CASE _Scenario OF
	QUEUE_CLEANUP_TEST_SCENARIO.REPEATED_EXECUTE_FAILURE:
		_Child.CleanupFailures := 2;
		_ExpectedExecuteFailures := 3;

	QUEUE_CLEANUP_TEST_SCENARIO.CANCEL_REQUEST_FAILURE:
		_Child.CancelFailures := 2;
		_ExpectedCancelFailures := 2;

	QUEUE_CLEANUP_TEST_SCENARIO.MESSAGE_FORMATTING_FAILURE:
		_ExpectedFailureMessage := "Task 'queue' processing failed";
END_CASE

_Resource.SetChild(child := _Child);
_Resource.SetThrowOnStartRelease(throwOnStartRelease := _InjectReleaseFailure);
_Queue.SetResourceManager(resourceManager := _Resource);
_Queue.StopWhenNoPendingTasks := TRUE;
_Queue.Enqueue(task := _Child);
_Queue.Enqueue(task := _Waiting);
Assert.ThatBool(actual := _Queue.Start(), message := "Prepared queue must accept Start").IsTrue();
END_METHOD

(*!
<summary>Advances one queue call and observes the selected failure or reuse case.</summary>
<description>
An escaping exception uses the framework's ExecuteTest diagnostic and proceeds to AfterTest.
</description>
*)
METHOD PROTECTED ExecuteTest : TOF_Testing.TEST_CYCLE_RESULT
ExecuteTest := TOF_Testing.TEST_CYCLE_RESULT.DONE;

IF CycleCount - _RunStartCycle > _MaxRunCycles THEN
	RecordFailure(message := "Queue cleanup or reuse exceeded its cycle budget");
	RETURN;
END_IF

_Queue.Execute();

CASE _Phase OF
	QUEUE_CLEANUP_TEST_PHASE.REUSE_RUN:
		IF _Queue.State.Stopped THEN
			checkSuccessfulReuse();
		ELSE
			ExecuteTest := TOF_Testing.TEST_CYCLE_RESULT.BUSY;
		END_IF

	QUEUE_CLEANUP_TEST_PHASE.OBSERVE_FAILED_RELEASE:
		Assert.ThatBool(
			actual := _Queue.State.Stopped AND_THEN _Queue.FinalStopReason.Failure,
			message := "Failed release must leave the queue stopped"
		).IsTrue();
		Assert.ThatUInt(
			actual := _Resource.ReleaseCalls,
			message := "A stopped queue must not retry a failed release"
		).ToBe(expected := 1);
		Assert.ThatBool(
			actual := _Resource.ResourceAcquired,
			message := "The failed release must leave the synthetic resource held"
		).IsTrue();

	QUEUE_CLEANUP_TEST_PHASE.FAILURE_RUN:
		IF NOT _Queue.State.Stopped THEN
			IF _Child.ExecuteFailuresRaised > 0 THEN
				observePendingFailure();
			END_IF

			ExecuteTest := TOF_Testing.TEST_CYCLE_RESULT.BUSY;
			RETURN;
		END_IF

		checkFailedRun();

		IF Outcome = TOF_Testing.TEST_OUTCOME.FAILED THEN
			RETURN;
		END_IF

		IF _Scenario = QUEUE_CLEANUP_TEST_SCENARIO.DELAYED_CLEANUP_AND_REUSE THEN
			IF startReuse() THEN
				_Phase := QUEUE_CLEANUP_TEST_PHASE.REUSE_RUN;
				_RunStartCycle := CycleCount;
				ExecuteTest := TOF_Testing.TEST_CYCLE_RESULT.BUSY;
			END_IF
		ELSIF _InjectReleaseFailure THEN
			_Phase := QUEUE_CLEANUP_TEST_PHASE.OBSERVE_FAILED_RELEASE;
			ExecuteTest := TOF_Testing.TEST_CYCLE_RESULT.BUSY;
		END_IF
END_CASE
END_METHOD

(*!
<summary>Checks ownership while the failed current child is still running.</summary>
<description>
On the initial failure call, confirms cleanup was deferred and optionally requests owner cancellation.
For held cleanup, counts subsequent queue calls before allowing the child to finish.
</description>
*)
METHOD PRIVATE observePendingFailure
IF NOT _Child.State.Running THEN
	RETURN;
END_IF

Assert.ThatBool(
	actual := _Queue.State.Running AND_THEN _Queue.RunningSubstate.Stopping,
	message := "The queue must wait in STOPPING for the child"
).IsTrue();
Assert.ThatBool(
	actual := _Resource.ResourceAcquired,
	message := "The queue must retain its resource during child cleanup"
).IsTrue();
Assert.ThatUInt(
	actual := _Resource.ReleaseCalls,
	message := "Release must wait for child cleanup"
).ToBe(expected := 0);
Assert.ThatBool(
	actual := _Waiting.State.Ready,
	message := "Waiting child must remain READY during cleanup"
).IsTrue();

IF NOT _FirstFailureObserved THEN
	_FirstFailureObserved := TRUE;
	Assert.ThatBool(
		actual := _Queue.OriginalStopReason.Failure,
		message := "The initial Execute exception must set the original result to FAILURE"
	).IsTrue();
	Assert.ThatUInt(
		actual := _Child.CompletedCleanupSteps,
		message := "The call that failed must not advance child cleanup"
	).ToBe(expected := 0);

	IF _RequestExternalCancel THEN
		Assert.ThatWideString(
			actual := _Queue.OriginalStopReason.Message,
			message := "Observe the first child failure before owner cancellation"
		).ToBe(expected := _ExpectedFailureMessage);
		Assert.ThatBool(
			actual := _Queue.Cancel(),
			message := "Owner Cancel must be accepted while failure cleanup is pending"
		).IsTrue();
		Assert.ThatBool(
			actual := _Queue.OriginalStopReason.ExternalCancel,
			message := "Accepted Cancel must replace the original failure reason"
		).IsTrue();
	END_IF

	RETURN;
END_IF

IF _Child.HoldCleanup THEN
	_HeldCycles := _HeldCycles + 1;
	Assert.ThatUInt(
		actual := _Child.CompletedCleanupSteps,
		message := "Held cleanup must not advance"
	).ToBe(expected := 0);

	IF _HeldCycles = _HeldObservationCycles THEN
		_Child.HoldCleanup := FALSE;
	END_IF
END_IF
END_METHOD

(*!
<summary>Checks the stopped queue, fault counts, entry ownership and release ordering.</summary>
*)
METHOD PRIVATE checkFailedRun
Assert.ThatBool(
	actual := _FirstFailureObserved,
	message := "Observe the initial failure while the child is RUNNING"
).IsTrue();
Assert.ThatBool(
	actual := _Child.State.Stopped,
	message := "Parent must not stop ahead of the failed child"
).IsTrue();
Assert.ThatUInt(
	actual := _Child.ExecuteFailuresRaised,
	message := "The configured Execute faults must occur"
).ToBe(expected := _ExpectedExecuteFailures);
Assert.ThatUInt(
	actual := _Child.CancelFailuresRaised,
	message := "The configured Cancel faults must occur"
).ToBe(expected := _ExpectedCancelFailures);
Assert.ThatUInt(
	actual := _Child.CompletedCleanupSteps,
	message := "Child must perform all cooperative cleanup steps"
).ToBe(expected := 3);
Assert.ThatBool(
	actual := _Child.FinalStopReason.ExternalCancel,
	message := "Failed child must finish through cooperative cancellation"
).IsTrue();
Assert.ThatBool(actual := _Waiting.State.Ready, message := "Waiting child must remain READY").IsTrue();
Assert.ThatInt(
	actual := _Waiting.Counter,
	message := "Waiting child must never execute"
).ToBe(expected := TOF_Core.SignedInt16.ZERO);
Assert.ThatDInt(
	actual := _Queue.PendingTaskCount,
	message := "Failed current and waiting entries must remain queued"
).ToBe(expected := 2);
Assert.ThatUInt(
	actual := _Resource.ReleaseCalls,
	message := "Queue must request parent release exactly once"
).ToBe(expected := 1);
Assert.ThatBool(
	actual := _Resource.EarlyRelease,
	message := "Parent release must follow child cleanup"
).IsFalse();

IF _Scenario = QUEUE_CLEANUP_TEST_SCENARIO.HELD_CLEANUP THEN
	Assert.ThatUInt(
		actual := _HeldCycles,
		message := "Every held queue call must be observed before unblocking cleanup"
	).ToBe(expected := _HeldObservationCycles);
END_IF

IF _RequestExternalCancel THEN
	Assert.ThatBool(
		actual := _Queue.OriginalStopReason.ExternalCancel,
		message := "Owner cancellation must remain the original reason"
	).IsTrue();
	Assert.ThatWideString(
		actual := _Queue.OriginalStopReason.Message,
		message := "Original diagnostic must describe owner cancellation"
	).ToBe(expected := "Cancelled by external logic");
ELSE
	Assert.ThatBool(
		actual := _Queue.OriginalStopReason.Failure,
		message := "The first failure must remain the original reason"
	).IsTrue();
	Assert.ThatWideString(
		actual := _Queue.OriginalStopReason.Message,
		message := "Original diagnostic must retain the first failure"
	).ToBe(expected := _ExpectedFailureMessage);
END_IF

IF _InjectReleaseFailure THEN
	Assert.ThatBool(
		actual := _Queue.FinalStopReason.Failure,
		message := "Release failure must determine the final reason"
	).IsTrue();
	Assert.ThatWideString(
		actual := _Queue.FinalStopReason.Message,
		message := "Final diagnostic must identify the failed release"
	).ToBe(expected := "Parent release failure");
	Assert.ThatBool(
		actual := _Resource.ResourceAcquired,
		message := "Failed release must leave the synthetic resource held"
	).IsTrue();
ELSIF _RequestExternalCancel THEN
	Assert.ThatBool(
		actual := _Queue.FinalStopReason.ExternalCancel,
		message := "Successful release must preserve the owner cancellation"
	).IsTrue();
	Assert.ThatWideString(
		actual := _Queue.FinalStopReason.Message,
		message := "Final diagnostic must retain the owner cancellation"
	).ToBe(expected := "Cancelled by external logic");
ELSE
	Assert.ThatBool(
		actual := _Queue.FinalStopReason.Failure,
		message := "Successful release must preserve the first failure"
	).IsTrue();
	Assert.ThatWideString(
		actual := _Queue.FinalStopReason.Message,
		message := "Later cleanup must not replace the first diagnostic"
	).ToBe(expected := _ExpectedFailureMessage);
END_IF

IF NOT _InjectReleaseFailure THEN
	Assert.ThatBool(actual := _Resource.ResourceAcquired, message := "Parent release must finish").IsFalse();
END_IF
END_METHOD

(*!
<summary>Resets the stopped queue and requeues its former failed child without fault injection.</summary>
*)
METHOD PRIVATE startReuse : BOOL
IF NOT _Queue.Reset() THEN
	RecordFailure(message := "Stopped queue must accept Reset before reuse");
	RETURN;
END_IF

Assert.ThatBool(actual := _Queue.State.Ready, message := "Reset must return the queue to READY").IsTrue();
Assert.ThatDInt(
	actual := _Queue.PendingTaskCount,
	message := "Reset must remove both retained entries"
).ToBe(expected := 0);
Assert.ThatWideString(
	actual := _Queue.OriginalStopReason.Message,
	message := "Reset must clear the original diagnostic"
).ToBe(expected := "");
Assert.ThatWideString(
	actual := _Queue.FinalStopReason.Message,
	message := "Reset must clear the final diagnostic"
).ToBe(expected := "");
Assert.ThatBool(
	actual := _Child.State.Stopped,
	message := "Queue Reset must not reset its borrowed child"
).IsTrue();

IF NOT _Queue.State.Ready OR_ELSE _Queue.PendingTaskCount <> 0 OR_ELSE NOT _Child.Reset() THEN
	RecordFailure(message := "Queue and child must be prepared before re-enqueueing");
	RETURN;
END_IF

_Child.ThrowOnFirstExecute := FALSE;
_Queue.Enqueue(task := _Child);
startReuse := _Queue.Start();
Assert.ThatBool(actual := startReuse, message := "Reset queue must accept a second Start").IsTrue();
END_METHOD

(*!
<summary>Verifies normal queue and child completion after resetting the failure run.</summary>
*)
METHOD PRIVATE checkSuccessfulReuse
Assert.ThatBool(
	actual := _Child.State.Stopped AND_THEN _Child.FinalStopReason.WorkDone,
	message := "Reused child must finish normally"
).IsTrue();
Assert.ThatBool(
	actual := _Queue.OriginalStopReason.WorkDone AND_THEN _Queue.FinalStopReason.WorkDone,
	message := "Reused queue must finish normally"
).IsTrue();
Assert.ThatUInt(
	actual := _Child.ExecuteFailuresRaised,
	message := "The reused child must have no Execute faults"
).ToBe(expected := 0);
Assert.ThatDInt(
	actual := _Queue.PendingTaskCount,
	message := "The successful reused queue must be empty"
).ToBe(expected := 0);
Assert.ThatUInt(
	actual := _Resource.ReleaseCalls,
	message := "Each run must request release once"
).ToBe(expected := 2);
Assert.ThatBool(
	actual := _Resource.EarlyRelease,
	message := "Reuse must also release after child completion"
).IsFalse();
Assert.ThatBool(actual := _Resource.ResourceAcquired, message := "Reuse must finish release").IsFalse();
Assert.ThatWideString(
	actual := _Queue.OriginalStopReason.Message,
	message := "Original diagnostics must not remain after reuse"
).ToBe(expected := "");
END_METHOD

(*!
<summary>Drains active synthetic work and clears the stopped fixtures before reporting.</summary>
<description>
Releases a deliberate child hold, then performs bounded cancellation using only synchronous synthetic fixtures.
Does not reset children or discard synthetic resource state while work remains active.
</description>
*)
METHOD PROTECTED AfterTest
VAR
	i : INT;
END_VAR
_Child.HoldCleanup := FALSE;

__TRY
	IF _Queue.State.Running THEN
		IF NOT _Queue.OriginalStopReason.ExternalCancel AND_THEN NOT _Queue.RunningSubstate.ResourceReleasing THEN
			_Queue.Cancel();
		END_IF

		FOR i := 1 TO _DrainBudget DO
			IF NOT _Queue.State.Running THEN
				EXIT;
			END_IF

			_Queue.Execute();
		END_FOR
	END_IF
__CATCH
	reportCleanupFailure(message := "An exception interrupted synthetic queue cancellation or drain");
__ENDTRY

IF _Queue.State.Running OR_ELSE _Child.State.Running OR_ELSE _Waiting.State.Running THEN
	reportCleanupFailure(message := "Synthetic queue cleanup left active work");
	RETURN;
END_IF

IF _Queue.State.Stopped THEN
	IF NOT _Queue.Reset() THEN
		reportCleanupFailure(message := "Stopped queue refused cleanup Reset");
		RETURN;
	END_IF
ELSE
	_Queue.ClearWaitingTasks();
END_IF

IF NOT _Queue.State.Ready OR_ELSE _Queue.PendingTaskCount <> 0 THEN
	reportCleanupFailure(message := "Queue must be READY and empty before resetting its former children");
	RETURN;
END_IF

IF NOT _Child.Reset() THEN
	reportCleanupFailure(message := "Synthetic current child refused cleanup Reset");
END_IF

IF NOT _Waiting.Reset() THEN
	reportCleanupFailure(message := "Synthetic waiting child refused cleanup Reset");
END_IF

_Resource.ResetFixture();
END_METHOD

(*!
<summary>Records a cleanup failure while preserving any earlier scenario diagnostic.</summary>
<description>Writes a separate ADS error when the test already has a recorded failure.</description>
<param name="message">Cleanup diagnostic copied during the call.</param>
*)
METHOD PRIVATE reportCleanupFailure
VAR_IN_OUT CONSTANT
	message : TOF_Core.ERROR_MESSAGE;
END_VAR
VAR
	logText : STRING(255);
END_VAR
IF Outcome = TOF_Testing.TEST_OUTCOME.FAILED THEN
	logText := TO_STRING(TOF_Core.WideStrings.ConcatFit255(Name, " cleanup: ", TO_WSTRING(message)));
	Tc2_System.ADSLOGSTR(
		msgCtrlMask := Tc2_System.Global_Variables.ADSLOG_MSGTYPE_ERROR,
		msgFmtStr := '%s',
		strArg := logText
	);
ELSE
	RecordFailure(message := message);
END_IF
END_METHOD

//! <summary>Borrows the concrete class name. Callers must not modify it.</summary>
{attribute 'monitoring' := 'call'}
PROPERTY ClassName : REFERENCE TO STRING
GET
ClassName REF= _ClassName;
END_GET
END_PROPERTY

//! <summary>Borrows the compiler-initialized namespace name. Callers must not modify it.</summary>
{attribute 'monitoring' := 'call'}
PROPERTY NamespaceName : REFERENCE TO STRING
GET
NamespaceName REF= CurrentNamespace.Name;
END_GET
END_PROPERTY

//! <summary>Reports the complete concrete instance size in bytes.</summary>
{attribute 'monitoring' := 'call'}
PROPERTY SelfSize : ULINT
GET
SelfSize := XSIZEOF(THIS^);
END_GET
END_PROPERTY

END_FUNCTION_BLOCK

// ---- Tests/Tasks/QueueCleanup/QueueCleanupQueue.TcPOU
(*
SPDX-FileCopyrightText: © 2026 Oleksandr Tiutyk <trofimich@gmail.com>
SPDX-License-Identifier: MIT
License: https://opensource.org/license/mit
*)

(*!
<summary>Supplies TaskQueue with an observable synthetic parent resource.</summary>
<description>
All queue execution and cancellation logic is inherited from the production TaskQueue. Bind a resource manager
through SetResourceManager before Start and keep the binding unchanged throughout the run. The scenario owns
the resource manager and children; the queue borrows them. Reset preserves the binding.
</description>
*)

FUNCTION_BLOCK QueueCleanupQueue EXTENDS TOF_Tasks.TaskQueue
VAR_STAT
	//! <summary>Class name shared by all instances of this function block.</summary>
	_ClassName : STRING := __POUNAME();
END_VAR
VAR
	//! <summary>Borrowed scenario resource manager; remains bound across queue resets.</summary>
	_ResourceManager : TOF_Core.IResourceManager;
END_VAR

{attribute 'monitoring' := 'call'}
PROPERTY ClassName : REFERENCE TO STRING
GET
ClassName REF= _ClassName;
END_GET
END_PROPERTY

(*!
<summary>Adds a live READY child through the production queue API.</summary>
<description>
Borrows the child without resetting or deleting it; it must be unique in this queue.
</description>
<param name="task">Live READY child whose lifecycle is delegated to the queue.</param>
*)
METHOD Enqueue
VAR_INPUT
	task : TOF_Tasks.ITask;
END_VAR
EnqueueTask(task := task);
END_METHOD

(*!
<summary>Borrows the test library namespace.</summary>
*)

{attribute 'monitoring' := 'call'}
PROPERTY NamespaceName : REFERENCE TO STRING
GET
NamespaceName REF= CurrentNamespace.Name;
END_GET
END_PROPERTY

(*!
<summary>Returns the resource manager supplied by the scenario.</summary>
<description>
Side-effect-free access. The scenario keeps the manager alive and the binding unchanged throughout the run.
</description>
*)

{attribute 'monitoring' := 'call'}
PROPERTY ResourceManager : TOF_Core.IResourceManager
GET
ResourceManager := _ResourceManager;
END_GET
END_PROPERTY

(*!
<summary>Binds the scenario's resource manager to the queue.</summary>
<description>
Call before Start and keep the binding unchanged throughout the run. The manager is borrowed; its owner must
keep it alive while bound. This method only assigns the binding and does not reset the queue or manager. Queue
Reset preserves the binding and the manager's observations.
</description>
<param name="resourceManager">Resource manager owned by the scenario.</param>
*)
METHOD INTERNAL SetResourceManager
VAR_INPUT
	resourceManager : TOF_Core.IResourceManager;
END_VAR
_ResourceManager := resourceManager;
END_METHOD

(*!
<summary>Reports the concrete fixture size.</summary>
*)

{attribute 'monitoring' := 'call'}
PROPERTY SelfSize : ULINT
GET
SelfSize := XSIZEOF(THIS^);
END_GET
END_PROPERTY

END_FUNCTION_BLOCK

// ---- Tests/Tasks/QueueCleanup/QueueCleanupResource.TcPOU
(*
SPDX-FileCopyrightText: © 2026 Oleksandr Tiutyk <trofimich@gmail.com>
SPDX-License-Identifier: MIT
License: https://opensource.org/license/mit
*)

(*!
<summary>Observes parent resource release without using a real resource.</summary>
<description>
Configure Child and ThrowOnStartRelease through SetChild and SetThrowOnStartRelease before the queue starts.
Child is borrowed and must outlive this manager. Acquisition takes one Execute; release takes two.
EarlyRelease records any request while Child is RUNNING. ReleaseCalls and EarlyRelease are observations only.
ResetFixture clears the synthetic state between independent test runs. No physical resource is created.
</description>
*)

FUNCTION_BLOCK QueueCleanupResource EXTENDS TOF_Core.Object IMPLEMENTS TOF_Core.IResourceManager
VAR_OUTPUT
	//! <summary>Borrowed child whose RUNNING state must prevent parent release.</summary>
	Child : TOF_Tasks.ITask;
	//! <summary>Raise a terminal release-attempt error on StartRelease.</summary>
	ThrowOnStartRelease : BOOL;
	//! <summary>Total StartRelease calls; read-only to tests.</summary>
	ReleaseCalls : UINT;
	//! <summary>Records whether release was requested while Child was RUNNING.</summary>
	EarlyRelease : BOOL;
END_VAR
VAR CONSTANT
	//! <summary>Execute calls required to complete synthetic release after its request.</summary>
	_ReleaseSteps : UINT := 2;
END_VAR
VAR_STAT
	//! <summary>Class name shared by all instances of this function block.</summary>
	_ClassName : STRING := __POUNAME();
END_VAR
VAR
	_Acquired : BOOL;
	_Acquiring : BOOL;
	_Releasing : BOOL;
	_ReleaseProgress : UINT;
END_VAR

{attribute 'monitoring' := 'call'}
PROPERTY ClassName : REFERENCE TO STRING
GET
ClassName REF= _ClassName;
END_GET
END_PROPERTY

(*!
<summary>Advances one synthetic acquisition or release step.</summary>
<description>
Idle calls do nothing; all operations are bounded and perform no I/O.
</description>
*)
METHOD Execute
IF _Acquiring THEN
	_Acquired := TRUE;
	_Acquiring := FALSE;
ELSIF _Releasing THEN
	_ReleaseProgress := _ReleaseProgress + 1;

	IF _ReleaseProgress >= _ReleaseSteps THEN
		_Acquired := FALSE;
		_Releasing := FALSE;
	END_IF
END_IF
END_METHOD

(*!
<summary>Returns this live fixture as the borrowed synthetic resource.</summary>
<description>
No real handle is created. The caller must not delete the returned object.
</description>
*)
METHOD GetResource : TOF_Core.IObject
GetResource := THIS^;
END_METHOD

(*!
<summary>Borrows the test library namespace.</summary>
*)

{attribute 'monitoring' := 'call'}
PROPERTY NamespaceName : REFERENCE TO STRING
GET
NamespaceName REF= CurrentNamespace.Name;
END_GET
END_PROPERTY

(*!
<summary>Reports whether the synthetic resource is held.</summary>
<description>
Has no side effects and does not throw.
</description>
*)

{attribute 'monitoring' := 'call'}
PROPERTY ResourceAcquired : BOOL
GET
ResourceAcquired := _Acquired;
END_GET
END_PROPERTY

(*!
<summary>Reports the concrete fixture size.</summary>
*)

{attribute 'monitoring' := 'call'}
PROPERTY SelfSize : ULINT
GET
SelfSize := XSIZEOF(THIS^);
END_GET
END_PROPERTY

(*!
<summary>Restores an idle synthetic resource and clears its observations.</summary>
<description>
Call only after the owning queue and children have stopped or before they start. Keeps the borrowed child
binding. Clears simulated state even after an injected terminal release error. Performs no physical release.
</description>
*)
METHOD INTERNAL ResetFixture
_Acquired := FALSE;
_Acquiring := FALSE;
_Releasing := FALSE;
_ReleaseProgress := 0;
ReleaseCalls := 0;
EarlyRelease := FALSE;
ThrowOnStartRelease := FALSE;
END_METHOD

(*!
<summary>Sets the child observed during resource release.</summary>
<description>
Call before the queue starts. The child is borrowed and must outlive the resource manager.
</description>
<param name="child">Child whose RUNNING state is observed during release.</param>
*)
METHOD INTERNAL SetChild
VAR_INPUT
	child : TOF_Tasks.ITask;
END_VAR
THIS^.Child := child;
END_METHOD

(*!
<summary>Configures the resource's release failure injection.</summary>
<description>
Call before the queue starts. Changes only the failure setting; resource progress and observations are
preserved.
</description>
<param name="throwOnStartRelease">Whether StartRelease raises the synthetic release-attempt error.</param>
*)
METHOD INTERNAL SetThrowOnStartRelease
VAR_INPUT
	throwOnStartRelease : BOOL;
END_VAR
THIS^.ThrowOnStartRelease := throwOnStartRelease;
END_METHOD

(*!
<summary>Requests synthetic acquisition completed by the next Execute.</summary>
<description>
Called once per acquire phase. Does nothing when already acquired.
</description>
*)
METHOD StartAcquire
IF NOT _Acquired THEN
	_Acquiring := TRUE;
END_IF
END_METHOD

(*!
<summary>Records release ordering and starts synthetic release.</summary>
<description>
Records EarlyRelease before optionally throwing. A thrown release deliberately leaves ResourceAcquired TRUE;
this models a failed terminal attempt without holding any real resource.
</description>
*)
METHOD StartRelease
VAR
	failure : TOF_Core.StandardException;
END_VAR
ReleaseCalls := ReleaseCalls + 1;

IF Child <> 0 AND_THEN Child.State.Running THEN
	EarlyRelease := TRUE;
END_IF

IF ThrowOnStartRelease THEN
	failure.Throw(
		sourceNamespaceName := NamespaceName,
		sourceClassName := ClassName,
		sourcePOUName := __POUNAME(),
		sourcePosition := __POSITION(),
		message := "Parent release failure"
	);
END_IF

_ReleaseProgress := 0;
_Releasing := TRUE;
END_METHOD

END_FUNCTION_BLOCK

// ---- Tests/Tasks/QueueCleanup/QueueCleanupChild.TcPOU
(*
SPDX-FileCopyrightText: © 2026 Oleksandr Tiutyk <trofimich@gmail.com>
SPDX-License-Identifier: MIT
License: https://opensource.org/license/mit
*)

(*!
<summary>Models a child whose Execute can throw while its lifecycle remains RUNNING.</summary>
<description>
Test-only implementation of ITask, independent of the base Task exception handler. It deliberately lets
Execute and Cancel exceptions reach the parent queue while remaining RUNNING. Deriving from Task would contain
these faults inside the child and would not exercise the queue's handling of a throwing ITask. Use Task
descendants for ordinary lifecycle tests; this fixture models the interface failure boundary. One owner drives
it. Configure inputs before Start; HoldCleanup may be cleared between calls to release the artificial hold.
Cancellation needs three successful Execute steps; injected cleanup failures do not count as steps. Public
outputs are observations only. Uses no hardware; exceptions are cleaned at the PLC task boundary.
</description>
*)

FUNCTION_BLOCK QueueCleanupChild EXTENDS TOF_Core.Object IMPLEMENTS TOF_Tasks.ITask
VAR_INPUT
	//! <summary>Inject one exception on the first Execute of a run.</summary>
	ThrowOnFirstExecute : BOOL := TRUE;
	//! <summary>When ThrowOnFirstExecute is enabled, use an exception whose GetMessage throws another exception.</summary>
	ThrowOnGetMessage : BOOL;
	//! <summary>Number of cleanup Execute calls that throw before successful cleanup steps.</summary>
	CleanupFailures : UINT;
	//! <summary>Number of cancellation requests that throw before accepting a request.</summary>
	CancelFailures : UINT;
	//! <summary>Keep accepted cancellation pending until the test releases this hold.</summary>
	HoldCleanup : BOOL;
END_VAR
VAR_OUTPUT
	//! <summary>Successful cleanup steps since the last Reset; read-only to tests.</summary>
	CompletedCleanupSteps : UINT;
	//! <summary>Exceptions raised by Execute in this run, including the initial fault.</summary>
	ExecuteFailuresRaised : UINT;
	//! <summary>Exceptions raised before accepting Cancel in this run.</summary>
	CancelFailuresRaised : UINT;
END_VAR
VAR CONSTANT
	//! <summary>Successful Execute calls required to finish synthetic cancellation.</summary>
	_CleanupSteps : UINT := 3;
END_VAR
VAR_STAT
	//! <summary>Class name shared by all instances of this function block.</summary>
	_ClassName : STRING := __POUNAME();
END_VAR
VAR
	_Name : WSTRING := TO_WSTRING(__POUNAME());
	_State : TOF_Tasks.TASK_STATE;
	_StateChanged : BOOL;
	_Substate : TOF_Tasks.TASK_RUNNING_SUBSTATE := TOF_Tasks.TASK_RUNNING_SUBSTATE.PROCESSING;
	_Reason : TOF_Tasks.TASK_STOP_REASON;
	_Message : TOF_Core.ERROR_MESSAGE;
	_StateView : TOF_Tasks.TaskState(_State, _StateChanged);
	_SubstateView : TOF_Tasks.TaskRunningSubstate(_Substate);
	_ReasonView : TOF_Tasks.TaskStopReason(_Reason, _Message);

	_InitialExecuteExceptionRaised : BOOL;
	_CancelRequested : BOOL;
	_CleanupFailuresLeft : UINT;
	_CancelFailuresLeft : UINT;
END_VAR

(*!
<summary>Injects configured request failures, then accepts cooperative cancellation.</summary>
<description>
Injected failures occur before acceptance and leave RUNNING intact. Repeated accepted cancellation refuses.
Acceptance selects STOPPING. Completion still requires Execute; no cleanup is performed by this method.
</description>
<param name="refuseReason">Reason for refusal; meaningful on FALSE.</param>
*)
METHOD Cancel : BOOL
VAR_OUTPUT
	refuseReason : TOF_Core.ERROR_MESSAGE;
END_VAR
VAR
	failure : TOF_Core.StandardException;
END_VAR
IF _State <> TOF_Tasks.TASK_STATE.RUNNING OR_ELSE _CancelRequested THEN
	refuseReason := "Fixture is not running or cancellation is already pending";
	RETURN;
END_IF

IF _CancelFailuresLeft > 0 THEN
	_CancelFailuresLeft := _CancelFailuresLeft - 1;
	CancelFailuresRaised := CancelFailuresRaised + 1;
	failure.Throw(
		sourceNamespaceName := NamespaceName,
		sourceClassName := ClassName,
		sourcePOUName := __POUNAME(),
		sourcePosition := __POSITION(),
		message := "Cancel request failure"
	);
END_IF

_CancelRequested := TRUE;
_Substate := TOF_Tasks.TASK_RUNNING_SUBSTATE.STOPPING;
_Reason := TOF_Tasks.TASK_STOP_REASON.EXTERNAL_CANCEL;
_Message := "Child cancellation requested";
Cancel := TRUE;
END_METHOD

{attribute 'monitoring' := 'call'}
PROPERTY ClassName : REFERENCE TO STRING
GET
ClassName REF= _ClassName;
END_GET
END_PROPERTY

(*!
<summary>Raises the initial fault or advances synthetic cancellation by one step.</summary>
<description>
An injected exception leaves RUNNING intact. Without ThrowOnFirstExecute, the first Execute completes
normally. After a fault, ordinary execution waits for an accepted Cancel; cleanup may throw or remain held.
</description>
*)
METHOD Execute
VAR
	failure : TOF_Core.StandardException;
	exceptionWithThrowingGetMessage : ThrowingGetMessageException;
END_VAR
_StateChanged := FALSE;

IF _State <> TOF_Tasks.TASK_STATE.RUNNING THEN
	RETURN;
END_IF

IF ThrowOnFirstExecute AND_THEN NOT _InitialExecuteExceptionRaised THEN
	_InitialExecuteExceptionRaised := TRUE;
	ExecuteFailuresRaised := ExecuteFailuresRaised + 1;

	IF ThrowOnGetMessage THEN
		exceptionWithThrowingGetMessage.Throw(
			sourceNamespaceName := NamespaceName,
			sourceClassName := ClassName,
			sourcePOUName := __POUNAME(),
			sourcePosition := __POSITION(),
			message := "First child failure"
		);
	ELSE
		failure.Throw(
			sourceNamespaceName := NamespaceName,
			sourceClassName := ClassName,
			sourcePOUName := __POUNAME(),
			sourcePosition := __POSITION(),
			message := "First child failure"
		);
	END_IF
END_IF

IF _CancelRequested THEN
	IF _CleanupFailuresLeft > 0 THEN
		_CleanupFailuresLeft := _CleanupFailuresLeft - 1;
		ExecuteFailuresRaised := ExecuteFailuresRaised + 1;
		failure.Throw(
			sourceNamespaceName := NamespaceName,
			sourceClassName := ClassName,
			sourcePOUName := __POUNAME(),
			sourcePosition := __POSITION(),
			message := "Later cleanup failure"
		);
	END_IF

	IF HoldCleanup THEN
		RETURN;
	END_IF

	CompletedCleanupSteps := CompletedCleanupSteps + 1;

	IF CompletedCleanupSteps < _CleanupSteps THEN
		RETURN;
	END_IF

	_Reason := TOF_Tasks.TASK_STOP_REASON.EXTERNAL_CANCEL;
	_Message := "Child cancellation completed";
ELSIF ThrowOnFirstExecute THEN
	RETURN;
ELSE
	_Reason := TOF_Tasks.TASK_STOP_REASON.WORK_DONE;
	_Message := "";
END_IF

_State := TOF_Tasks.TASK_STATE.STOPPED;
_StateChanged := TRUE;
END_METHOD

(*!
<summary>Borrows the synthetic termination result.</summary>
<description>
The fixture has no separate release failure, so both result views share backing fields. Observe only.
</description>
*)

{attribute 'monitoring' := 'call'}
PROPERTY FinalStopReason : REFERENCE TO TOF_Tasks.TaskStopReason
GET
FinalStopReason REF= _ReasonView;
END_GET
END_PROPERTY

(*!
<summary>Borrows the fixture display name.</summary>
<description>
Read-only storage valid while the fixture lives.
</description>
*)

{attribute 'monitoring' := 'call'}
PROPERTY Name : REFERENCE TO WSTRING
GET
Name REF= _Name;
END_GET
END_PROPERTY

(*!
<summary>Borrows the test library namespace.</summary>
*)

{attribute 'monitoring' := 'call'}
PROPERTY NamespaceName : REFERENCE TO STRING
GET
NamespaceName REF= CurrentNamespace.Name;
END_GET
END_PROPERTY

(*!
<summary>Borrows the synthetic termination result.</summary>
<description>
The fixture has no separate release failure, so both result views share backing fields. Observe only.
</description>
*)

{attribute 'monitoring' := 'call'}
PROPERTY OriginalStopReason : REFERENCE TO TOF_Tasks.TaskStopReason
GET
OriginalStopReason REF= _ReasonView;
END_GET
END_PROPERTY

(*!
<summary>Clears a stopped fixture for reuse without changing its configuration.</summary>
<description>
READY is a successful no-op; RUNNING refuses. Clears observations, pending faults and result text, and
restores the initial PROCESSING substate for reuse.
</description>
<param name="refuseReason">Reason for refusal; meaningful on FALSE.</param>
*)
METHOD Reset : BOOL
VAR_OUTPUT
	refuseReason : TOF_Core.ERROR_MESSAGE;
END_VAR
IF _State = TOF_Tasks.TASK_STATE.RUNNING THEN
	refuseReason := "Fixture is still RUNNING";
	RETURN;
END_IF

IF _State = TOF_Tasks.TASK_STATE.READY THEN
	Reset := TRUE;
	RETURN;
END_IF

_State := TOF_Tasks.TASK_STATE.READY;
_Substate := TOF_Tasks.TASK_RUNNING_SUBSTATE.PROCESSING;
_StateChanged := TRUE;
_Reason := TOF_Tasks.TASK_STOP_REASON.WORK_DONE;
_Message := "";
_InitialExecuteExceptionRaised := FALSE;
_CancelRequested := FALSE;
_CleanupFailuresLeft := 0;
_CancelFailuresLeft := 0;
CompletedCleanupSteps := 0;
ExecuteFailuresRaised := 0;
CancelFailuresRaised := 0;
Reset := TRUE;
END_METHOD

(*!
<summary>Returns zero because the child has no managed resource.</summary>
*)

{attribute 'monitoring' := 'call'}
PROPERTY ResourceManager : TOF_Core.IResourceManager
GET
END_GET
END_PROPERTY

(*!
<summary>Borrows the synthetic processing phase.</summary>
<description>
Meaningful only while RUNNING. No real resource is acquired.
</description>
*)

{attribute 'monitoring' := 'call'}
PROPERTY RunningSubstate : REFERENCE TO TOF_Tasks.TaskRunningSubstate
GET
RunningSubstate REF= _SubstateView;
END_GET
END_PROPERTY

(*!
<summary>Reports the concrete fixture size.</summary>
*)

{attribute 'monitoring' := 'call'}
PROPERTY SelfSize : ULINT
GET
SelfSize := XSIZEOF(THIS^);
END_GET
END_PROPERTY

(*!
<summary>Starts a READY fixture and copies the fault-injection settings.</summary>
<description>
Does not execute work. A non-READY call refuses without changing state.
</description>
<param name="refuseReason">Reason for refusal; meaningful on FALSE.</param>
*)
METHOD Start : BOOL
VAR_OUTPUT
	refuseReason : TOF_Core.ERROR_MESSAGE;
END_VAR
IF _State <> TOF_Tasks.TASK_STATE.READY THEN
	refuseReason := "Fixture is not READY";
	RETURN;
END_IF

_CleanupFailuresLeft := CleanupFailures;
_CancelFailuresLeft := CancelFailures;
_State := TOF_Tasks.TASK_STATE.RUNNING;
_StateChanged := TRUE;
Start := TRUE;
END_METHOD

(*!
<summary>Borrows the live synthetic lifecycle state.</summary>
<description>
Observe only; the fixture must outlive this view.
</description>
*)

{attribute 'monitoring' := 'call'}
PROPERTY State : REFERENCE TO TOF_Tasks.TaskState
GET
State REF= _StateView;
END_GET
END_PROPERTY

END_FUNCTION_BLOCK

// ---- Tests/Tasks/Stopping/TimerTimingTestGroup.TcPOU
(*
SPDX-FileCopyrightText: © 2026 Oleksandr Tiutyk <trofimich@gmail.com>
SPDX-License-Identifier: MIT
License: https://opensource.org/license/mit
*)

(*!
<summary>Groups timer timing, lifecycle and restart scenarios.</summary>
<description>
Owns the test cases and their fixed child array. Use from a single PLC task and keep the group at a stable address.
</description>
*)

{attribute 'no_assign'}
{attribute 'no_explicit_call' := 'do not call this function block directly'}
FUNCTION_BLOCK TimerTimingTestGroup EXTENDS TOF_Testing.TestGroup<13>
VAR_STAT
	{attribute 'hide'}
	_ClassName : STRING := __POUNAME();
END_VAR
VAR
	_PositiveIntervalSameCallRestart : TimerCompletionPulseTest(
		name := "PositiveIntervalSameCallRestart",
		parent := THIS^,
		interval := T#30MS
	);
	_ZeroIntervalSameCallRestart : TimerCompletionPulseTest(
		name := "ZeroIntervalSameCallRestart",
		parent := THIS^,
		interval := TOF_Core.Times.MIN_VALUE
	);
	_DefaultNameAndMetadata : TimerMetadataTest(
		name := "DefaultNameAndMetadata",
		parent := THIS^
	);
	_CancelBeforeFirstExecuteAndReuse : TimerCancelBeforeExecuteTest(
		name := "CancelBeforeFirstExecuteAndReuse",
		parent := THIS^
	);
	_ResetAfterCompletion : TimerResetAfterCompletionTest(
		name := "ResetAfterCompletion",
		parent := THIS^
	);
	_IntervalAssignmentPreservesObservation : TimerIntervalObservationTest(
		name := "IntervalAssignmentPreservesObservation",
		parent := THIS^
	);
	_RestartWaitsForStopping : TimerPendingRestartTest(
		name := "RestartWaitsForStopping",
		parent := THIS^
	);
	_RestartPreservesIntervalOnResetFailure : TimerRestartResetFailureTest(
		name := "RestartPreservesIntervalOnResetFailure",
		parent := THIS^
	);
	_RestartRetainsIntervalOnStartFailure : TimerRestartStartFailureTest(
		name := "RestartRetainsIntervalOnStartFailure",
		parent := THIS^
	);
	_CompletionCallbackCanReset : TimerCompletionCallbackTest(
		name := "CompletionCallbackCanReset",
		parent := THIS^
	);
	_DelayedFirstExecuteUsesStartAnchor : DelayedTimerObservationTest(
		name := "DelayedFirstExecuteUsesStartAnchor",
		parent := THIS^,
		scenario := DELAYED_TIMER_TEST_SCENARIO.AFTER_START
	);
	_CancelAfterUnobservedExpiry : DelayedTimerObservationTest(
		name := "CancelAfterUnobservedExpiry",
		parent := THIS^,
		scenario := DELAYED_TIMER_TEST_SCENARIO.CANCEL_BEFORE_EXECUTE
	);
	_PositiveRestartUsesStartAnchor : DelayedTimerObservationTest(
		name := "PositiveRestartUsesStartAnchor",
		parent := THIS^,
		scenario := DELAYED_TIMER_TEST_SCENARIO.AFTER_ACTIVE_RESTART
	);

	_Children : ARRAY [0.._ChildCount - 1] OF TOF_Testing.ITestElement :=
	[
		_PositiveIntervalSameCallRestart,
		_ZeroIntervalSameCallRestart,
		_DefaultNameAndMetadata,
		_CancelBeforeFirstExecuteAndReuse,
		_ResetAfterCompletion,
		_IntervalAssignmentPreservesObservation,
		_RestartWaitsForStopping,
		_RestartPreservesIntervalOnResetFailure,
		_RestartRetainsIntervalOnStartFailure,
		_CompletionCallbackCanReset,
		_DelayedFirstExecuteUsesStartAnchor,
		_CancelAfterUnobservedExpiry,
		_PositiveRestartUsesStartAnchor
	];
END_VAR

//! <summary>Borrows the fixed child array. Callers must not modify it.</summary>
{attribute 'monitoring' := 'call'}
PROPERTY Children : REFERENCE TO ARRAY [0.._ChildCount - 1] OF TOF_Testing.ITestElement
GET
Children REF= _Children;
END_GET
END_PROPERTY

//! <summary>Borrows the concrete class name. Callers must not modify it.</summary>
{attribute 'monitoring' := 'call'}
PROPERTY ClassName : REFERENCE TO STRING
GET
ClassName REF= _ClassName;
END_GET
END_PROPERTY

//! <summary>Borrows the compiler-initialized namespace. Callers must not modify it.</summary>
{attribute 'monitoring' := 'call'}
PROPERTY NamespaceName : REFERENCE TO STRING
GET
NamespaceName REF= CurrentNamespace.Name;
END_GET
END_PROPERTY

//! <summary>Reports the concrete instance size in bytes.</summary>
{attribute 'monitoring' := 'call'}
PROPERTY SelfSize : ULINT
GET
SelfSize := XSIZEOF(THIS^);
END_GET
END_PROPERTY

END_FUNCTION_BLOCK

// ---- Tests/Tasks/Stopping/TimerCompletionPulseTest.TcPOU
(*
SPDX-FileCopyrightText: © 2026 Oleksandr Tiutyk <trofimich@gmail.com>
SPDX-License-Identifier: MIT
License: https://opensource.org/license/mit
*)

(*!
<summary>Checks repeated timer completion, immediate restart and pulse clearing.</summary>
<description>
The zero preset must finish on its first Execute. For a positive preset, compares completion against the
independent task timestamp, the actual observation gap and a millisecond of preset precision. Time must
advance normally. One task owns the persistent timer and AfterTest prepares it for another run.
</description>
*)

{attribute 'no_assign'}
{attribute 'no_explicit_call' := 'do not call this function block directly'}
FUNCTION_BLOCK TimerCompletionPulseTest EXTENDS TOF_Testing.MultiCycleTest
VAR_STAT
	{attribute 'hide'}
	_ClassName : STRING := __POUNAME();
END_VAR
VAR CONSTANT
	//! <summary>Task clock counts 100 ns per tick.</summary>
	_TaskTimeTicksPerMillisecond : ULINT := 10000;
	//! <summary>Accounts for the millisecond precision of the TIME preset.</summary>
	_TimingToleranceTicks : ULINT := 10000;
	//! <summary>Multiple runs expose stale TON observations and restart state.</summary>
	_RunCount : UINT := 3;
END_VAR
VAR
	_Timer : TOF_Timers.Timer(name := "Completion pulse timer");
	_Interval : TIME;
	_CompletedRuns : UINT;
	_StartedAt : ULINT;
	_LastObservedAt : ULINT;
END_VAR

(*!
<summary>Selects the case configuration and its ten-second nominal deadline.</summary>
<param name="name">Display name of this case.</param>
<param name="parent">Group that owns this test.</param>
<param name="interval">Zero or positive preset under test.</param>
*)
METHOD FB_init : BOOL
VAR_INPUT
	bInitRetains: BOOL; // TRUE: the retain variables are initialized (reset warm / reset cold)
	bInCopyCode: BOOL; // TRUE: the instance will be copied to the copy code afterward (online change)
	name : WSTRING;
	parent : TOF_Testing.ITestElement;
	interval : TIME;
END_VAR
_Interval := interval;
_Timeout := T#10S;
FB_init := TRUE;
END_METHOD

(*!
<summary>Configures the timer and records the independent start timestamp.</summary>
*)
METHOD PROTECTED BeforeTest
_CompletedRuns := 0;
_Timer.Interval := _Interval;
_StartedAt := Tc2_System.F_GetTaskTime();
_LastObservedAt := _StartedAt;

IF NOT _Timer.Start() THEN
	RecordFailure(message := "Prepared timer must accept Start");
	RETURN;
END_IF

Assert.ThatBool(
	actual := _Timer.Triggered,
	message := "Start must leave the completion pulse clear"
).IsFalse();
END_METHOD

(*!
<summary>Advances one timer call per cycle and restarts in the cycle that observes completion.</summary>
*)
METHOD PROTECTED ExecuteTest : TOF_Testing.TEST_CYCLE_RESULT
VAR
	elapsed : BOOL;
END_VAR
ExecuteTest := TOF_Testing.TEST_CYCLE_RESULT.DONE;
_Timer.Execute();

IF _CompletedRuns = _RunCount THEN
	Assert.ThatBool(
		actual := _Timer.Triggered,
		message := "The next Execute must clear the completion pulse"
	).IsFalse();
	Assert.ThatBool(
		actual := _Timer.Elapsed,
		message := "Idle Execute must preserve elapsed until Reset"
	).IsTrue();
	Assert.ThatBool(actual := _Timer.State.Stopped, message := "Idle Execute must preserve STOPPED").IsTrue();

	RETURN;
END_IF

elapsed := _Timer.Elapsed;

IF _Interval = TOF_Core.Times.MIN_VALUE THEN
	Assert.ThatBool(actual := elapsed, message := "Zero interval must set TON.Q on its first Execute").IsTrue();
ELSE
	checkPositiveTiming(triggered := _Timer.Triggered);
END_IF

Assert.ThatBool(
	actual := _Timer.Triggered,
	message := "Triggered must match the newly observed TON.Q in the same Execute"
).ToBe(expected := elapsed);

IF Outcome = TOF_Testing.TEST_OUTCOME.FAILED THEN
	RETURN;
END_IF

IF _Timer.Triggered THEN
	Assert.ThatBool(
		actual := _Timer.Triggered,
		message := "Repeated getter reads must preserve the completion pulse"
	).IsTrue();
	Assert.ThatBool(
		actual := _Timer.State.Stopped,
		message := "Timer must already be STOPPED on completion"
	).IsTrue();
	Assert.ThatBool(
		actual := _Timer.FinalStopReason.WorkDone,
		message := "Natural timer completion must report WORK_DONE"
	).IsTrue();
	Assert.ThatBool(
		actual := _Timer.ElapsedTime = _Interval,
		message := "Completed elapsed time must equal the preset"
	).IsTrue();

	_CompletedRuns := _CompletedRuns + 1;

	IF _CompletedRuns < _RunCount THEN
		_StartedAt := Tc2_System.F_GetTaskTime();
		_LastObservedAt := _StartedAt;

		IF NOT _Timer.Restart() THEN
			RecordFailure(message := "Restart must succeed in the completion cycle");
			RETURN;
		END_IF

		Assert.ThatBool(
			actual := _Timer.State.Running,
			message := "Restart must begin a new run immediately"
		).IsTrue();
		Assert.ThatBool(actual := _Timer.Elapsed, message := "Restart must reset the old TON.Q").IsFalse();
		Assert.ThatBool(actual := _Timer.Triggered, message := "Restart must clear the consumed pulse").IsFalse();
	END_IF
ELSE
	Assert.ThatBool(actual := _Timer.State.Running, message := "An incomplete timer must remain RUNNING").IsTrue();
END_IF

ExecuteTest := TOF_Testing.TEST_CYCLE_RESULT.BUSY;
END_METHOD

(*!
<summary>Compares a positive completion with independent task time.</summary>
<description>
Accepts the elapsed time at the first eligible observation within the time quantization allowance.
</description>
<param name="triggered">Completion pulse observed after the current Execute.</param>
*)
METHOD PRIVATE checkPositiveTiming
VAR_INPUT
	triggered : BOOL;
END_VAR
VAR
	currentTaskTime : ULINT;
	elapsedTicks : ULINT;
	observationGap : ULINT;
	presetTicks : ULINT;
END_VAR
currentTaskTime := Tc2_System.F_GetTaskTime();

IF currentTaskTime < _LastObservedAt THEN
	RecordFailure(message := "Independent task time moved backwards");
	RETURN;
END_IF

elapsedTicks := currentTaskTime - _StartedAt;
observationGap := currentTaskTime - _LastObservedAt;
_LastObservedAt := currentTaskTime;
presetTicks := TO_ULINT(_Interval) * _TaskTimeTicksPerMillisecond;

IF triggered THEN
	Assert.ThatBool(
		actual := elapsedTicks + _TimingToleranceTicks >= presetTicks,
		message := "Positive timer must not complete ahead of the preset"
	).IsTrue();
	Assert.ThatBool(
		actual := elapsedTicks <= presetTicks + observationGap + _TimingToleranceTicks,
		message := "Completion must occur at the first eligible observation"
	).IsTrue();
ELSE
	Assert.ThatBool(
		actual := elapsedTicks <= presetTicks + _TimingToleranceTicks,
		message := "The timer must trigger at the first observation past its preset"
	).IsTrue();
END_IF
END_METHOD

(*!
<summary>Returns the owned timer to READY before reporting the result.</summary>
<description>
Cooperatively cancels active work and clears any retained TON observations through Reset.
</description>
*)
METHOD PROTECTED AfterTest
Assert.ThatBool(
	actual := PrepareTimerTestForReuse(timer := _Timer),
	message := "The timer must return to READY after cleanup"
).IsTrue();
END_METHOD

//! <summary>Borrows the concrete class name. Callers must not modify it.</summary>
{attribute 'monitoring' := 'call'}
PROPERTY ClassName : REFERENCE TO STRING
GET
ClassName REF= _ClassName;
END_GET
END_PROPERTY

//! <summary>Borrows the compiler-initialized namespace. Callers must not modify it.</summary>
{attribute 'monitoring' := 'call'}
PROPERTY NamespaceName : REFERENCE TO STRING
GET
NamespaceName REF= CurrentNamespace.Name;
END_GET
END_PROPERTY

//! <summary>Reports the concrete instance size in bytes.</summary>
{attribute 'monitoring' := 'call'}
PROPERTY SelfSize : ULINT
GET
SelfSize := XSIZEOF(THIS^);
END_GET
END_PROPERTY

END_FUNCTION_BLOCK

// ---- Tests/Tasks/Stopping/PrepareTimerTestForReuse.TcPOU
(*
SPDX-FileCopyrightText: © 2026 Oleksandr Tiutyk <trofimich@gmail.com>
SPDX-License-Identifier: MIT
License: https://opensource.org/license/mit
*)

(*!
<summary>Returns a resource-free timer fixture to READY.</summary>
<description>
Call after disabling any injected callback failure or stopping hold. Advances pending cancellation once.
Returns FALSE if the fixture still needs work or refuses Reset. Owns no resource or exception state.
</description>
<param name="timer">Live timer fixture owned by the calling test.</param>
*)
FUNCTION PrepareTimerTestForReuse : BOOL
VAR_INPUT
	timer : TOF_Tasks.ITask;
END_VAR

IF timer.State.Running THEN
	IF NOT timer.OriginalStopReason.ExternalCancel THEN
		timer.Cancel();
	END_IF

	timer.Execute();
END_IF

IF timer.State.Stopped THEN
	IF NOT timer.Reset() THEN
		RETURN;
	END_IF
END_IF

PrepareTimerTestForReuse := timer.State.Ready;

END_FUNCTION

// ---- Tests/Tasks/Stopping/TimerMetadataTest.TcPOU
(*
SPDX-FileCopyrightText: © 2026 Oleksandr Tiutyk <trofimich@gmail.com>
SPDX-License-Identifier: MIT
License: https://opensource.org/license/mit
*)

(*!
<summary>Checks default and explicit names before Start and after reuse.</summary>
<description>
The case executes in one PLC callback with a persistent timer and no external resources.
AfterTest prepares the fixture for reuse by the runner.
</description>
*)

{attribute 'no_assign'}
{attribute 'no_explicit_call' := 'do not call this function block directly'}
FUNCTION_BLOCK TimerMetadataTest EXTENDS TOF_Testing.SingleCycleTest
VAR_STAT
	{attribute 'hide'}
	_ClassName : STRING := __POUNAME();
END_VAR
VAR
	_Timer : TOF_Timers.Timer(name := "");
	_NamedTimer : TOF_Timers.Timer(name := "Explicit timer");
END_VAR

(*!
<summary>Checks default and explicit names before Start and after reuse.</summary>
*)
METHOD PROTECTED ExecuteTest
VAR
	initialName : WSTRING;
	borrowedName : REFERENCE TO WSTRING;
	nameAfterReset : REFERENCE TO WSTRING;
END_VAR
borrowedName REF= _Timer.Name;

IF NOT __ISVALIDREF(borrowedName) THEN
	RecordFailure(message := "Timer must expose a valid borrowed name");
	RETURN;
END_IF

initialName := borrowedName;
Assert.ThatBool(
	actual := Tc2_Standard.WLEFT(STR := initialName, SIZE := Tc2_Standard.WLEN(STR := "Timer")) = "Timer",
	message := "Default name must contain the initialized Timer class before Start"
).IsTrue();
Assert.ThatBool(
	actual := _NamedTimer.Name = "Explicit timer",
	message := "Explicit name must be copied unchanged"
).IsTrue();
Assert.ThatBool(
	actual := _Timer.ClassName = 'Timer',
	message := "ClassName must identify the concrete Timer"
).IsTrue();
Assert.ThatBool(
	actual := _Timer.NamespaceName = 'TOF_Timers',
	message := "NamespaceName must identify the timer library"
).IsTrue();
Assert.ThatBool(
	actual := _Timer.SelfSize = XSIZEOF(_Timer),
	message := "SelfSize must match the concrete timer"
).IsTrue();
Assert.ThatBool(actual := _Timer.State.Ready, message := "Metadata reads must not start the timer").IsTrue();
_Timer.Interval := TOF_Core.Times.MIN_VALUE;

IF NOT _Timer.Start() THEN
	RecordFailure(message := "Unnamed timer must accept Start");
	RETURN;
END_IF

_Timer.Execute();
Assert.ThatBool(actual := _Timer.Triggered, message := "Unnamed zero timer must complete").IsTrue();

IF NOT _Timer.Reset() THEN
	RecordFailure(message := "Completed unnamed timer must accept Reset");
	RETURN;
END_IF

nameAfterReset REF= _Timer.Name;

IF NOT __ISVALIDREF(nameAfterReset) THEN
	RecordFailure(message := "Reset must leave the borrowed name reference valid");
	RETURN;
END_IF

Assert.ThatBool(
	actual := ADR(nameAfterReset) = ADR(borrowedName) AND_THEN nameAfterReset = initialName,
	message := "The name storage must survive Reset"
).IsTrue();
END_METHOD

(*!
<summary>Returns the owned timer to READY before reporting the result.</summary>
<description>
Cooperatively cancels active work and clears any retained TON observations through Reset.
</description>
*)
METHOD PROTECTED AfterTest
Assert.ThatBool(
	actual := PrepareTimerTestForReuse(timer := _Timer),
	message := "The timer must return to READY after cleanup"
).IsTrue();
END_METHOD

//! <summary>Borrows the concrete class name. Callers must not modify it.</summary>
{attribute 'monitoring' := 'call'}
PROPERTY ClassName : REFERENCE TO STRING
GET
ClassName REF= _ClassName;
END_GET
END_PROPERTY

//! <summary>Borrows the compiler-initialized namespace. Callers must not modify it.</summary>
{attribute 'monitoring' := 'call'}
PROPERTY NamespaceName : REFERENCE TO STRING
GET
NamespaceName REF= CurrentNamespace.Name;
END_GET
END_PROPERTY

//! <summary>Reports the concrete instance size in bytes.</summary>
{attribute 'monitoring' := 'call'}
PROPERTY SelfSize : ULINT
GET
SelfSize := XSIZEOF(THIS^);
END_GET
END_PROPERTY

END_FUNCTION_BLOCK

// ---- Tests/Tasks/Stopping/TimerCancelBeforeExecuteTest.TcPOU
(*
SPDX-FileCopyrightText: © 2026 Oleksandr Tiutyk <trofimich@gmail.com>
SPDX-License-Identifier: MIT
License: https://opensource.org/license/mit
*)

(*!
<summary>Checks cancellation before the first Execute and reuse after reset.</summary>
<description>
The case executes in one PLC callback with a persistent timer and no external resources.
AfterTest prepares the fixture for reuse by the runner.
</description>
*)

{attribute 'no_assign'}
{attribute 'no_explicit_call' := 'do not call this function block directly'}
FUNCTION_BLOCK TimerCancelBeforeExecuteTest EXTENDS TOF_Testing.SingleCycleTest
VAR_STAT
	{attribute 'hide'}
	_ClassName : STRING := __POUNAME();
END_VAR
VAR CONSTANT
	//! <summary>Keeps the old timer active until the scenario cancels or restarts it.</summary>
	_ActiveInterval : TIME := T#1H;
END_VAR
VAR
	_Timer : TOF_Timers.Timer(name := "Cancel timer");
END_VAR

(*!
<summary>Checks cancellation before the first Execute and reuse after reset.</summary>
*)
METHOD PROTECTED ExecuteTest
_Timer.Interval := _ActiveInterval;

IF NOT _Timer.Start() THEN
	RecordFailure(message := "Long timer must accept Start");
	RETURN;
END_IF

Assert.ThatBool(actual := _Timer.Reset(), message := "Reset must refuse a running timer").IsFalse();

IF NOT _Timer.Cancel() THEN
	RecordFailure(message := "Cancellation must be accepted before the first Execute");
	RETURN;
END_IF

Assert.ThatBool(actual := _Timer.Cancel(), message := "Repeated cancellation must be refused").IsFalse();
_Timer.Execute();
Assert.ThatBool(
	actual := _Timer.State.Stopped,
	message := "Ordinary cancellation must finish in one Execute"
).IsTrue();
Assert.ThatBool(
	actual := _Timer.FinalStopReason.ExternalCancel,
	message := "Cancellation must remain the final reason"
).IsTrue();
Assert.ThatBool(
	actual := _Timer.Triggered,
	message := "Cancellation must not become successful completion"
).IsFalse();
Assert.ThatBool(actual := _Timer.Elapsed, message := "Cancelled long timer must not report elapsed").IsFalse();

IF NOT _Timer.Reset() THEN
	RecordFailure(message := "Cancelled timer must accept Reset");
	RETURN;
END_IF

Assert.ThatBool(
	actual := _Timer.ElapsedTime = TOF_Core.Times.MIN_VALUE,
	message := "Reset must clear elapsed time"
).IsTrue();
Assert.ThatBool(
	actual := _Timer.Interval = _ActiveInterval,
	message := "Reset must preserve the configured interval"
).IsTrue();

IF NOT _Timer.SetIntervalAndRestart(interval := TOF_Core.Times.MIN_VALUE) THEN
	RecordFailure(message := "Cancelled timer must support immediate reuse");
	RETURN;
END_IF

_Timer.Execute();
Assert.ThatBool(actual := _Timer.Triggered, message := "Reused timer must complete normally").IsTrue();
END_METHOD

(*!
<summary>Returns the owned timer to READY before reporting the result.</summary>
<description>
Cooperatively cancels active work and clears any retained TON observations through Reset.
</description>
*)
METHOD PROTECTED AfterTest
Assert.ThatBool(
	actual := PrepareTimerTestForReuse(timer := _Timer),
	message := "The timer must return to READY after cleanup"
).IsTrue();
END_METHOD

//! <summary>Borrows the concrete class name. Callers must not modify it.</summary>
{attribute 'monitoring' := 'call'}
PROPERTY ClassName : REFERENCE TO STRING
GET
ClassName REF= _ClassName;
END_GET
END_PROPERTY

//! <summary>Borrows the compiler-initialized namespace. Callers must not modify it.</summary>
{attribute 'monitoring' := 'call'}
PROPERTY NamespaceName : REFERENCE TO STRING
GET
NamespaceName REF= CurrentNamespace.Name;
END_GET
END_PROPERTY

//! <summary>Reports the concrete instance size in bytes.</summary>
{attribute 'monitoring' := 'call'}
PROPERTY SelfSize : ULINT
GET
SelfSize := XSIZEOF(THIS^);
END_GET
END_PROPERTY

END_FUNCTION_BLOCK

// ---- Tests/Tasks/Stopping/TimerResetAfterCompletionTest.TcPOU
(*
SPDX-FileCopyrightText: © 2026 Oleksandr Tiutyk <trofimich@gmail.com>
SPDX-License-Identifier: MIT
License: https://opensource.org/license/mit
*)

(*!
<summary>Checks repeated Execute and explicit Reset after natural completion.</summary>
<description>
The case executes in one PLC callback with a persistent timer and no external resources.
AfterTest prepares the fixture for reuse by the runner.
</description>
*)

{attribute 'no_assign'}
{attribute 'no_explicit_call' := 'do not call this function block directly'}
FUNCTION_BLOCK TimerResetAfterCompletionTest EXTENDS TOF_Testing.SingleCycleTest
VAR_STAT
	{attribute 'hide'}
	_ClassName : STRING := __POUNAME();
END_VAR
VAR
	_Timer : TOF_Timers.Timer(name := "Completed timer");
END_VAR

(*!
<summary>Checks repeated Execute and explicit Reset after natural completion.</summary>
*)
METHOD PROTECTED ExecuteTest
_Timer.Interval := TOF_Core.Times.MIN_VALUE;

IF NOT _Timer.Start() THEN
	RecordFailure(message := "Zero timer must accept Start");
	RETURN;
END_IF

_Timer.Execute();
Assert.ThatBool(actual := _Timer.Triggered, message := "First Execute must expose completion").IsTrue();
Assert.ThatBool(actual := _Timer.Start(), message := "Start must refuse STOPPED without Reset").IsFalse();
Assert.ThatBool(actual := _Timer.Cancel(), message := "Cancel must refuse an already completed timer").IsFalse();
_Timer.Execute();
Assert.ThatBool(
	actual := _Timer.Triggered,
	message := "A second Execute in the same cycle must clear the pulse"
).IsFalse();
Assert.ThatBool(actual := _Timer.Elapsed, message := "Idle Execute must preserve retained elapsed").IsTrue();
Assert.ThatBool(
	actual := _Timer.FinalStopReason.WorkDone,
	message := "Idle Execute must preserve the result"
).IsTrue();

IF NOT _Timer.Reset() THEN
	RecordFailure(message := "Completed timer must accept Reset");
	RETURN;
END_IF

Assert.ThatBool(actual := _Timer.State.Ready, message := "Successful Reset must restore READY").IsTrue();
Assert.ThatBool(actual := _Timer.Elapsed, message := "Reset must clear retained elapsed").IsFalse();
Assert.ThatBool(actual := _Timer.Triggered, message := "Reset must clear the completion pulse").IsFalse();
Assert.ThatBool(
	actual := _Timer.ElapsedTime = TOF_Core.Times.MIN_VALUE,
	message := "Reset must clear ET"
).IsTrue();

IF NOT _Timer.Restart() THEN
	RecordFailure(message := "Restart must also work from READY");
	RETURN;
END_IF

_Timer.Execute();
Assert.ThatBool(
	actual := _Timer.Triggered,
	message := "Restart after explicit Reset must yield a fresh completion"
).IsTrue();
END_METHOD

(*!
<summary>Returns the owned timer to READY before reporting the result.</summary>
<description>
Cooperatively cancels active work and clears any retained TON observations through Reset.
</description>
*)
METHOD PROTECTED AfterTest
Assert.ThatBool(
	actual := PrepareTimerTestForReuse(timer := _Timer),
	message := "The timer must return to READY after cleanup"
).IsTrue();
END_METHOD

//! <summary>Borrows the concrete class name. Callers must not modify it.</summary>
{attribute 'monitoring' := 'call'}
PROPERTY ClassName : REFERENCE TO STRING
GET
ClassName REF= _ClassName;
END_GET
END_PROPERTY

//! <summary>Borrows the compiler-initialized namespace. Callers must not modify it.</summary>
{attribute 'monitoring' := 'call'}
PROPERTY NamespaceName : REFERENCE TO STRING
GET
NamespaceName REF= CurrentNamespace.Name;
END_GET
END_PROPERTY

//! <summary>Reports the concrete instance size in bytes.</summary>
{attribute 'monitoring' := 'call'}
PROPERTY SelfSize : ULINT
GET
SelfSize := XSIZEOF(THIS^);
END_GET
END_PROPERTY

END_FUNCTION_BLOCK

// ---- Tests/Tasks/Stopping/TimerIntervalObservationTest.TcPOU
(*
SPDX-FileCopyrightText: © 2026 Oleksandr Tiutyk <trofimich@gmail.com>
SPDX-License-Identifier: MIT
License: https://opensource.org/license/mit
*)

(*!
<summary>Checks that changing the timer preset preserves the current observation.</summary>
<description>
Starts a long interval and waits for a nonzero elapsed observation before changing the preset in RUNNING.
Also checks assignment while READY and STOPPED. One task owns the timer and AfterTest prepares it for reuse.
</description>
*)

{attribute 'no_assign'}
{attribute 'no_explicit_call' := 'do not call this function block directly'}
FUNCTION_BLOCK TimerIntervalObservationTest EXTENDS TOF_Testing.MultiCycleTest
VAR_STAT
	{attribute 'hide'}
	_ClassName : STRING := __POUNAME();
END_VAR
VAR CONSTANT
	//! <summary>Keeps the old timer active until the scenario cancels or restarts it.</summary>
	_ActiveInterval : TIME := T#1H;
END_VAR
VAR
	_Timer : TOF_Timers.Timer(name := "Configured timer");
END_VAR

(*!
<summary>Sets the initial interval while READY and starts the timer explicitly.</summary>
*)
METHOD PROTECTED BeforeTest
_Timer.Interval := _ActiveInterval;
Assert.ThatBool(
	actual := _Timer.State.Ready,
	message := "Configuring Interval must leave a READY timer idle"
).IsTrue();
Assert.ThatBool(actual := _Timer.Start(), message := "The configured timer must accept Start").IsTrue();
END_METHOD

(*!
<summary>Changes the running preset after observing positive elapsed time.</summary>
*)
METHOD PROTECTED ExecuteTest : TOF_Testing.TEST_CYCLE_RESULT
VAR
	observedTime : TIME;
END_VAR
_Timer.Execute();
observedTime := _Timer.ElapsedTime;

IF observedTime = TOF_Core.Times.MIN_VALUE THEN
	ExecuteTest := TOF_Testing.TEST_CYCLE_RESULT.BUSY;
	RETURN;
END_IF

ExecuteTest := TOF_Testing.TEST_CYCLE_RESULT.DONE;
Assert.ThatBool(
	actual := _Timer.State.Running,
	message := "A nonzero elapsed observation must belong to a running timer"
).IsTrue();
_Timer.Interval := TOF_Core.Times.MIN_VALUE;
Assert.ThatBool(
	actual := _Timer.State.Running,
	message := "Assignment of the zero preset must preserve RUNNING"
).IsTrue();
Assert.ThatBool(
	actual := _Timer.ElapsedTime = observedTime,
	message := "Assignment must preserve the nonzero elapsed observation"
).IsTrue();
Assert.ThatBool(
	actual := _Timer.Elapsed,
	message := "Assignment must leave TON.Q at its previous value"
).IsFalse();
Assert.ThatBool(
	actual := _Timer.Triggered,
	message := "Assignment must leave the completion pulse clear"
).IsFalse();

_Timer.Execute();
Assert.ThatBool(
	actual := _Timer.Triggered,
	message := "The next Execute must evaluate the changed zero preset"
).IsTrue();
observedTime := _Timer.ElapsedTime;

_Timer.Interval := _ActiveInterval;
Assert.ThatBool(
	actual := _Timer.State.Stopped,
	message := "Assigning a preset while STOPPED must keep the timer stopped"
).IsTrue();
Assert.ThatBool(
	actual := _Timer.Elapsed,
	message := "Assignment in STOPPED must preserve retained TON.Q"
).IsTrue();
Assert.ThatBool(
	actual := _Timer.ElapsedTime = observedTime,
	message := "Assignment in STOPPED must preserve elapsed time"
).IsTrue();

_Timer.Execute();
Assert.ThatBool(
	actual := _Timer.Elapsed,
	message := "Stopped Execute must preserve the retained TON observation"
).IsTrue();

IF NOT _Timer.Reset() THEN
	RecordFailure(message := "Explicit Reset must remain available after assigning the preset");
	RETURN;
END_IF

Assert.ThatBool(actual := _Timer.Elapsed, message := "Explicit Reset must clear TON.Q").IsFalse();
END_METHOD

(*!
<summary>Returns the owned timer to READY before reporting the result.</summary>
<description>
Cooperatively cancels active work and clears any retained TON observations through Reset.
</description>
*)
METHOD PROTECTED AfterTest
Assert.ThatBool(
	actual := PrepareTimerTestForReuse(timer := _Timer),
	message := "The timer must return to READY after cleanup"
).IsTrue();
END_METHOD

//! <summary>Borrows the concrete class name. Callers must not modify it.</summary>
{attribute 'monitoring' := 'call'}
PROPERTY ClassName : REFERENCE TO STRING
GET
ClassName REF= _ClassName;
END_GET
END_PROPERTY

//! <summary>Borrows the compiler-initialized namespace. Callers must not modify it.</summary>
{attribute 'monitoring' := 'call'}
PROPERTY NamespaceName : REFERENCE TO STRING
GET
NamespaceName REF= CurrentNamespace.Name;
END_GET
END_PROPERTY

//! <summary>Reports the concrete instance size in bytes.</summary>
{attribute 'monitoring' := 'call'}
PROPERTY SelfSize : ULINT
GET
SelfSize := XSIZEOF(THIS^);
END_GET
END_PROPERTY

END_FUNCTION_BLOCK

// ---- Tests/Tasks/Stopping/TimerPendingRestartTest.TcPOU
(*
SPDX-FileCopyrightText: © 2026 Oleksandr Tiutyk <trofimich@gmail.com>
SPDX-License-Identifier: MIT
License: https://opensource.org/license/mit
*)

(*!
<summary>Checks one-step restart preparation while asynchronous stopping remains pending.</summary>
<description>
The case executes in one PLC callback with a persistent restart probe and no external resources.
AfterTest prepares the fixture for reuse by the runner.
</description>
*)

{attribute 'no_assign'}
{attribute 'no_explicit_call' := 'do not call this function block directly'}
FUNCTION_BLOCK TimerPendingRestartTest EXTENDS TOF_Testing.SingleCycleTest
VAR_STAT
	{attribute 'hide'}
	_ClassName : STRING := __POUNAME();
END_VAR
VAR CONSTANT
	//! <summary>Keeps the old timer active until the scenario cancels or restarts it.</summary>
	_ActiveInterval : TIME := T#1H;

	//! <summary>Positive interval selected for the replacement run.</summary>
	_PositiveInterval : TIME := T#30MS;
END_VAR
VAR
	_Timer : TimerRestartProbe(name := "Pending restart");
END_VAR

(*!
<summary>Checks one-step restart preparation while asynchronous stopping remains pending.</summary>
<description>Compares stopping calls relative to the cumulative count at entry.</description>
*)
METHOD PROTECTED ExecuteTest
VAR
	initialStoppingCalls : UINT;
END_VAR
initialStoppingCalls := _Timer.StoppingCalls;

_Timer.Interval := _ActiveInterval;
_Timer.AllowStopping := FALSE;

IF NOT _Timer.Start() THEN
	RecordFailure(message := "Probe must accept initial Start");
	RETURN;
END_IF

Assert.ThatBool(
	actual := _Timer.SetIntervalAndRestart(interval := _PositiveInterval),
	message := "Restart must refuse while stopping remains pending"
).IsFalse();
Assert.ThatBool(
	actual := _Timer.State.Running,
	message := "Refused preparation must retain active cleanup"
).IsTrue();
Assert.ThatBool(
	actual := _Timer.StoppingCalls = TO_UINT(TO_UDINT(initialStoppingCalls) + 1),
	message := "Preparation must advance stopping exactly once"
).IsTrue();
Assert.ThatBool(
	actual := _Timer.Interval = _ActiveInterval,
	message := "Pending stopping must preserve the old PT"
).IsTrue();
Assert.ThatBool(actual := _Timer.Restart(), message := "Another pending restart must also refuse").IsFalse();
Assert.ThatBool(
	actual := _Timer.StoppingCalls = TO_UINT(TO_UDINT(initialStoppingCalls) + 2),
	message := "Repeated preparation must add only one stopping call"
).IsTrue();
_Timer.AllowStopping := TRUE;
_Timer.Execute();
Assert.ThatBool(actual := _Timer.State.Stopped, message := "Open gate must allow cleanup to finish").IsTrue();
Assert.ThatBool(
	actual := _Timer.FinalStopReason.ExternalCancel,
	message := "Active restart preparation cancels the old run"
).IsTrue();
Assert.ThatBool(
	actual := _Timer.Interval = _ActiveInterval,
	message := "Finishing cleanup must not apply a deferred PT"
).IsTrue();
_Timer.Execute();
Assert.ThatBool(
	actual := _Timer.State.Stopped,
	message := "Refused restart must not schedule a later Start"
).IsTrue();

IF NOT _Timer.SetIntervalAndRestart(interval := _PositiveInterval) THEN
	RecordFailure(message := "An explicit retry must succeed after cleanup");
	RETURN;
END_IF

Assert.ThatBool(
	actual := _Timer.Interval = _PositiveInterval,
	message := "Successful retry must apply the new PT"
).IsTrue();

IF NOT _Timer.Cancel() THEN
	RecordFailure(message := "Scenario must cancel its active replacement run");
	RETURN;
END_IF

_Timer.Execute();
Assert.ThatBool(
	actual := _Timer.State.Stopped AND_THEN _Timer.FinalStopReason.ExternalCancel,
	message := "The replacement run must finish cancellation"
).IsTrue();
END_METHOD

(*!
<summary>Returns the owned timer to READY before reporting the result.</summary>
<description>
Reopens the stopping gate and disables callback injections before cooperative cleanup.
</description>
*)
METHOD PROTECTED AfterTest
_Timer.AllowStopping := TRUE;
_Timer.ThrowOnBeforeStart := FALSE;
_Timer.ThrowOnReset := FALSE;
_Timer.ResetOnAfterStop := FALSE;

Assert.ThatBool(
	actual := PrepareTimerTestForReuse(timer := _Timer),
	message := "The timer must return to READY after cleanup"
).IsTrue();
END_METHOD

//! <summary>Borrows the concrete class name. Callers must not modify it.</summary>
{attribute 'monitoring' := 'call'}
PROPERTY ClassName : REFERENCE TO STRING
GET
ClassName REF= _ClassName;
END_GET
END_PROPERTY

//! <summary>Borrows the compiler-initialized namespace. Callers must not modify it.</summary>
{attribute 'monitoring' := 'call'}
PROPERTY NamespaceName : REFERENCE TO STRING
GET
NamespaceName REF= CurrentNamespace.Name;
END_GET
END_PROPERTY

//! <summary>Reports the concrete instance size in bytes.</summary>
{attribute 'monitoring' := 'call'}
PROPERTY SelfSize : ULINT
GET
SelfSize := XSIZEOF(THIS^);
END_GET
END_PROPERTY

END_FUNCTION_BLOCK

// ---- Tests/Tasks/Stopping/TimerRestartProbe.TcPOU
(*
SPDX-FileCopyrightText: © 2026 Oleksandr Tiutyk <trofimich@gmail.com>
SPDX-License-Identifier: MIT
License: https://opensource.org/license/mit
*)

(*!
<summary>Exercises inherited timer restart contracts with controlled stopping and callback failures.</summary>
<description>
Owned persistently by one test scenario and driven by its task only. AllowStopping delays termination without
blocking. Exceptions deliberately injected outside FB lifecycle methods must be converted to refusal by Task;
the enclosing AutomationRunner supplies exception cleanup and the terminal allocation boundary.
</description>
*)

FUNCTION_BLOCK TimerRestartProbe EXTENDS TOF_Timers.Timer
VAR_INPUT
	//! <summary>Allows the next stopping call to finish; FALSE keeps cleanup pending.</summary>
	AllowStopping : BOOL := TRUE;
	//! <summary>Injects a start-preparation exception before the base timer is started.</summary>
	ThrowOnBeforeStart : BOOL;
	//! <summary>Injects a reset exception before the base TON state is cleared.</summary>
	ThrowOnReset : BOOL;
	//! <summary>Exercises the supported Reset callback after final completion.</summary>
	ResetOnAfterStop : BOOL;
END_VAR
VAR_OUTPUT
	//! <summary>Counts stopping calls so tests can detect extra advancement or busy waiting.</summary>
	StoppingCalls : UINT;
END_VAR
VAR_STAT
	_ProbeClassName : STRING := __POUNAME();
END_VAR
VAR
	_Failure : TOF_Core.StandardException;
END_VAR

(*!
<summary>Borrows the concrete fixture name from initialized static read-only storage.</summary>
*)
{attribute 'monitoring' := 'call'}
PROPERTY ClassName : REFERENCE TO STRING
GET
ClassName REF= _ProbeClassName;
END_GET
END_PROPERTY

(*!
<summary>Borrows the test library namespace; callers must not modify the text.</summary>
*)
{attribute 'monitoring' := 'call'}
PROPERTY NamespaceName : REFERENCE TO STRING
GET
NamespaceName REF= CurrentNamespace.Name;
END_GET
END_PROPERTY

(*!
<summary>Returns the size in bytes of the concrete restart fixture.</summary>
*)
{attribute 'monitoring' := 'call'}
PROPERTY SelfSize : ULINT
GET
SelfSize := XSIZEOF(THIS^);
END_GET
END_PROPERTY

(*!
<summary>Injects a refusal before preserving the base timer start preparation.</summary>
<description>The deliberate exception exercises Task.Start failure handling without leaving an active TON.</description>
*)
METHOD PROTECTED OnBeforeStart
IF ThrowOnBeforeStart THEN
	raiseConfiguredFailure(message := "Timer start preparation failure");
END_IF

SUPER^.OnBeforeStart();
END_METHOD

(*!
<summary>Injects a refusal before preserving the base TON reset.</summary>
<description>A refused reset leaves the old interval and elapsed observations available for assertions.</description>
*)
METHOD PROTECTED OnReset
IF ThrowOnReset THEN
	raiseConfiguredFailure(message := "Timer reset failure");
END_IF

SUPER^.OnReset();
END_METHOD

(*!
<summary>Counts one stopping step and combines base readiness with the configured gate.</summary>
<param name="readyToRelease">TRUE only when inherited stopping is complete and the test opens its gate.</param>
*)
METHOD PROTECTED OnStopping
VAR_OUTPUT
	readyToRelease : BOOL;
END_VAR
StoppingCalls := StoppingCalls + 1;
SUPER^.OnStopping(readyToRelease => readyToRelease);
readyToRelease := readyToRelease AND AllowStopping;
END_METHOD

(*!
<summary>Optionally resets the completed timer through the supported notification callback.</summary>
<description>Reset clears the completion observation before the outer Execute returns.</description>
*)
METHOD PROTECTED OnAfterStop
SUPER^.OnAfterStop();

IF ResetOnAfterStop THEN
	Reset();
END_IF
END_METHOD

(*!
<summary>Raises a diagnostic exception to exercise the inherited callback refusal boundary.</summary>
<description>Used only by operational hooks; never called from FB_init, FB_exit or FB_reinit.</description>
<param name="message">Diagnostic text copied into the synthetic exception.</param>
*)
METHOD PRIVATE raiseConfiguredFailure
VAR_INPUT
	message : WSTRING(255);
END_VAR
_Failure.Throw(
	sourceNamespaceName := NamespaceName,
	sourceClassName := ClassName,
	sourcePOUName := __POUNAME(),
	sourcePosition := __POSITION(),
	message := message
);
END_METHOD

END_FUNCTION_BLOCK

// ---- Tests/Tasks/Stopping/TimerRestartResetFailureTest.TcPOU
(*
SPDX-FileCopyrightText: © 2026 Oleksandr Tiutyk <trofimich@gmail.com>
SPDX-License-Identifier: MIT
License: https://opensource.org/license/mit
*)

(*!
<summary>Checks interval and observations when the reset hook refuses restart.</summary>
<description>
The case executes in one PLC callback with a persistent restart probe and no external resources.
AfterTest prepares the fixture for reuse by the runner.
</description>
*)

{attribute 'no_assign'}
{attribute 'no_explicit_call' := 'do not call this function block directly'}
FUNCTION_BLOCK TimerRestartResetFailureTest EXTENDS TOF_Testing.SingleCycleTest
VAR_STAT
	{attribute 'hide'}
	_ClassName : STRING := __POUNAME();
END_VAR
VAR CONSTANT
	//! <summary>Keeps the old timer active until the scenario cancels or restarts it.</summary>
	_ActiveInterval : TIME := T#1H;

	//! <summary>Positive interval selected for the replacement run.</summary>
	_PositiveInterval : TIME := T#30MS;
END_VAR
VAR
	_Timer : TimerRestartProbe(name := "Reset refusal");
END_VAR

(*!
<summary>Checks interval and observations when the reset hook refuses restart.</summary>
*)
METHOD PROTECTED ExecuteTest
_Timer.Interval := TOF_Core.Times.MIN_VALUE;

IF NOT _Timer.Start() THEN
	RecordFailure(message := "Probe must accept initial Start");
	RETURN;
END_IF

_Timer.Execute();
Assert.ThatBool(actual := _Timer.Triggered, message := "Old run must complete before reset injection").IsTrue();
_Timer.ThrowOnReset := TRUE;
Assert.ThatBool(
	actual := _Timer.SetIntervalAndRestart(interval := _PositiveInterval),
	message := "Reset exception must be converted to restart refusal"
).IsFalse();
Assert.ThatBool(actual := _Timer.State.Stopped, message := "Reset refusal must preserve STOPPED").IsTrue();
Assert.ThatBool(
	actual := _Timer.Interval = TOF_Core.Times.MIN_VALUE,
	message := "Failed preparation must preserve old PT"
).IsTrue();
Assert.ThatBool(actual := _Timer.Elapsed, message := "Failure before the base reset must retain old Q").IsTrue();
_Timer.ThrowOnReset := FALSE;

IF NOT _Timer.SetIntervalAndRestart(interval := _ActiveInterval) THEN
	RecordFailure(message := "Restart must recover after removing reset injection");
	RETURN;
END_IF

Assert.ThatBool(actual := _Timer.Elapsed, message := "Successful reset must clear old Q").IsFalse();
Assert.ThatBool(actual := _Timer.Triggered, message := "Successful restart must clear the old pulse").IsFalse();

IF NOT _Timer.Cancel() THEN
	RecordFailure(message := "Scenario must cancel the recovered run");
	RETURN;
END_IF

_Timer.Execute();
Assert.ThatBool(
	actual := _Timer.State.Stopped AND_THEN _Timer.FinalStopReason.ExternalCancel,
	message := "The replacement run must finish cancellation"
).IsTrue();
END_METHOD

(*!
<summary>Returns the owned timer to READY before reporting the result.</summary>
<description>
Reopens the stopping gate and disables callback injections before cooperative cleanup.
</description>
*)
METHOD PROTECTED AfterTest
_Timer.AllowStopping := TRUE;
_Timer.ThrowOnBeforeStart := FALSE;
_Timer.ThrowOnReset := FALSE;
_Timer.ResetOnAfterStop := FALSE;

Assert.ThatBool(
	actual := PrepareTimerTestForReuse(timer := _Timer),
	message := "The timer must return to READY after cleanup"
).IsTrue();
END_METHOD

//! <summary>Borrows the concrete class name. Callers must not modify it.</summary>
{attribute 'monitoring' := 'call'}
PROPERTY ClassName : REFERENCE TO STRING
GET
ClassName REF= _ClassName;
END_GET
END_PROPERTY

//! <summary>Borrows the compiler-initialized namespace. Callers must not modify it.</summary>
{attribute 'monitoring' := 'call'}
PROPERTY NamespaceName : REFERENCE TO STRING
GET
NamespaceName REF= CurrentNamespace.Name;
END_GET
END_PROPERTY

//! <summary>Reports the concrete instance size in bytes.</summary>
{attribute 'monitoring' := 'call'}
PROPERTY SelfSize : ULINT
GET
SelfSize := XSIZEOF(THIS^);
END_GET
END_PROPERTY

END_FUNCTION_BLOCK

// ---- Tests/Tasks/Stopping/TimerRestartStartFailureTest.TcPOU
(*
SPDX-FileCopyrightText: © 2026 Oleksandr Tiutyk <trofimich@gmail.com>
SPDX-License-Identifier: MIT
License: https://opensource.org/license/mit
*)

(*!
<summary>Checks the configured new interval after late start-preparation refusal.</summary>
<description>
The case executes in one PLC callback with a persistent restart probe and no external resources.
AfterTest prepares the fixture for reuse by the runner.
</description>
*)

{attribute 'no_assign'}
{attribute 'no_explicit_call' := 'do not call this function block directly'}
FUNCTION_BLOCK TimerRestartStartFailureTest EXTENDS TOF_Testing.SingleCycleTest
VAR_STAT
	{attribute 'hide'}
	_ClassName : STRING := __POUNAME();
END_VAR
VAR CONSTANT
	//! <summary>Positive interval selected for the replacement run.</summary>
	_PositiveInterval : TIME := T#30MS;
END_VAR
VAR
	_Timer : TimerRestartProbe(name := "Start refusal");
END_VAR

(*!
<summary>Checks the configured new interval after late start-preparation refusal.</summary>
*)
METHOD PROTECTED ExecuteTest
_Timer.Interval := TOF_Core.Times.MIN_VALUE;
_Timer.ThrowOnBeforeStart := TRUE;
Assert.ThatBool(
	actual := _Timer.SetIntervalAndRestart(interval := _PositiveInterval),
	message := "Start preparation exception must be converted to restart refusal"
).IsFalse();
Assert.ThatBool(
	actual := _Timer.State.Ready,
	message := "Refused Start must leave the prepared timer READY"
).IsTrue();
Assert.ThatBool(
	actual := _Timer.Interval = _PositiveInterval,
	message := "Late Start refusal must retain the new PT"
).IsTrue();
Assert.ThatBool(
	actual := _Timer.Elapsed,
	message := "Injected refusal before base Start must leave Q clear"
).IsFalse();
_Timer.Execute();
Assert.ThatBool(
	actual := _Timer.State.Ready,
	message := "Refused restart must not schedule automatic execution"
).IsTrue();
_Timer.ThrowOnBeforeStart := FALSE;

IF NOT _Timer.Start() THEN
	RecordFailure(message := "Explicit Start must recover after removing injection");
	RETURN;
END_IF

IF NOT _Timer.Cancel() THEN
	RecordFailure(message := "Scenario must cancel the recovered run");
	RETURN;
END_IF

_Timer.Execute();
Assert.ThatBool(
	actual := _Timer.State.Stopped AND_THEN _Timer.FinalStopReason.ExternalCancel,
	message := "The replacement run must finish cancellation"
).IsTrue();
END_METHOD

(*!
<summary>Returns the owned timer to READY before reporting the result.</summary>
<description>
Reopens the stopping gate and disables callback injections before cooperative cleanup.
</description>
*)
METHOD PROTECTED AfterTest
_Timer.AllowStopping := TRUE;
_Timer.ThrowOnBeforeStart := FALSE;
_Timer.ThrowOnReset := FALSE;
_Timer.ResetOnAfterStop := FALSE;

Assert.ThatBool(
	actual := PrepareTimerTestForReuse(timer := _Timer),
	message := "The timer must return to READY after cleanup"
).IsTrue();
END_METHOD

//! <summary>Borrows the concrete class name. Callers must not modify it.</summary>
{attribute 'monitoring' := 'call'}
PROPERTY ClassName : REFERENCE TO STRING
GET
ClassName REF= _ClassName;
END_GET
END_PROPERTY

//! <summary>Borrows the compiler-initialized namespace. Callers must not modify it.</summary>
{attribute 'monitoring' := 'call'}
PROPERTY NamespaceName : REFERENCE TO STRING
GET
NamespaceName REF= CurrentNamespace.Name;
END_GET
END_PROPERTY

//! <summary>Reports the concrete instance size in bytes.</summary>
{attribute 'monitoring' := 'call'}
PROPERTY SelfSize : ULINT
GET
SelfSize := XSIZEOF(THIS^);
END_GET
END_PROPERTY

END_FUNCTION_BLOCK

// ---- Tests/Tasks/Stopping/TimerCompletionCallbackTest.TcPOU
(*
SPDX-FileCopyrightText: © 2026 Oleksandr Tiutyk <trofimich@gmail.com>
SPDX-License-Identifier: MIT
License: https://opensource.org/license/mit
*)

(*!
<summary>Checks the documented completion observation when OnAfterStop resets the timer.</summary>
<description>
The case executes in one PLC callback with a persistent restart probe and no external resources.
AfterTest prepares the fixture for reuse by the runner.
</description>
*)

{attribute 'no_assign'}
{attribute 'no_explicit_call' := 'do not call this function block directly'}
FUNCTION_BLOCK TimerCompletionCallbackTest EXTENDS TOF_Testing.SingleCycleTest
VAR_STAT
	{attribute 'hide'}
	_ClassName : STRING := __POUNAME();
END_VAR
VAR
	_Timer : TimerRestartProbe(name := "Callback reset");
END_VAR

(*!
<summary>Checks the documented completion observation when OnAfterStop resets the timer.</summary>
*)
METHOD PROTECTED ExecuteTest
_Timer.ResetOnAfterStop := TRUE;
_Timer.Interval := TOF_Core.Times.MIN_VALUE;

IF NOT _Timer.Start() THEN
	RecordFailure(message := "Callback probe must accept Start");
	RETURN;
END_IF

Assert.ThatBool(
	actual := _Timer.State.Running,
	message := "Probe must be RUNNING before the completion callback"
).IsTrue();
_Timer.Execute();
Assert.ThatBool(actual := _Timer.State.Ready, message := "Supported callback Reset must restore READY").IsTrue();
Assert.ThatBool(
	actual := _Timer.Triggered,
	message := "Callback Reset may clear the pulse before Execute returns"
).IsFalse();
Assert.ThatBool(actual := _Timer.Elapsed, message := "Callback Reset must clear retained Q").IsFalse();
Assert.ThatBool(
	actual := _Timer.ElapsedTime = TOF_Core.Times.MIN_VALUE,
	message := "Callback Reset must clear ET"
).IsTrue();
END_METHOD

(*!
<summary>Returns the owned timer to READY before reporting the result.</summary>
<description>
Reopens the stopping gate and disables callback injections before cooperative cleanup.
</description>
*)
METHOD PROTECTED AfterTest
_Timer.AllowStopping := TRUE;
_Timer.ThrowOnBeforeStart := FALSE;
_Timer.ThrowOnReset := FALSE;
_Timer.ResetOnAfterStop := FALSE;

Assert.ThatBool(
	actual := PrepareTimerTestForReuse(timer := _Timer),
	message := "The timer must return to READY after cleanup"
).IsTrue();
END_METHOD

//! <summary>Borrows the concrete class name. Callers must not modify it.</summary>
{attribute 'monitoring' := 'call'}
PROPERTY ClassName : REFERENCE TO STRING
GET
ClassName REF= _ClassName;
END_GET
END_PROPERTY

//! <summary>Borrows the compiler-initialized namespace. Callers must not modify it.</summary>
{attribute 'monitoring' := 'call'}
PROPERTY NamespaceName : REFERENCE TO STRING
GET
NamespaceName REF= CurrentNamespace.Name;
END_GET
END_PROPERTY

//! <summary>Reports the concrete instance size in bytes.</summary>
{attribute 'monitoring' := 'call'}
PROPERTY SelfSize : ULINT
GET
SelfSize := XSIZEOF(THIS^);
END_GET
END_PROPERTY

END_FUNCTION_BLOCK

// ---- Tests/Tasks/Stopping/DelayedTimerObservationTest.TcPOU
(*
SPDX-FileCopyrightText: © 2026 Oleksandr Tiutyk <trofimich@gmail.com>
SPDX-License-Identifier: MIT
License: https://opensource.org/license/mit
*)

(*!
<summary>Checks how a positive timer behaves when its first Execute is intentionally delayed.</summary>
<description>
Uses independent task time to postpone the first observation until after the preset. Each case owns a
persistent timer for one PLC task. AfterTest returns the timer to READY.
</description>
*)

{attribute 'no_assign'}
{attribute 'no_explicit_call' := 'do not call this function block directly'}
FUNCTION_BLOCK DelayedTimerObservationTest EXTENDS TOF_Testing.MultiCycleTest
VAR_STAT
	{attribute 'hide'}
	_ClassName : STRING := __POUNAME();
END_VAR
VAR CONSTANT
	//! <summary>Positive preset that is observable across PLC cycles.</summary>
	_PositiveInterval : TIME := T#30MS;
	//! <summary>Task clock counts 100 ns per tick.</summary>
	_TaskTimeTicksPerMillisecond : ULINT := 10000;
	//! <summary>Accounts for the millisecond precision of the TIME preset.</summary>
	_TimingToleranceTicks : ULINT := 10000;

	//! <summary>Keeps the old timer active until the scenario cancels or restarts it.</summary>
	_ActiveInterval : TIME := T#1H;
END_VAR
VAR
	_Timer : TOF_Timers.Timer(name := "Delayed timer");
	_Scenario : DELAYED_TIMER_TEST_SCENARIO;
	_StartedAt : ULINT;
END_VAR

(*!
<summary>Selects the case configuration and its ten-second nominal deadline.</summary>
<param name="name">Display name of this case.</param>
<param name="parent">Group that owns this test.</param>
<param name="scenario">Operation to perform before the delayed observation.</param>
*)
METHOD FB_init : BOOL
VAR_INPUT
	bInitRetains: BOOL; // TRUE: the retain variables are initialized (reset warm / reset cold)
	bInCopyCode: BOOL; // TRUE: the instance will be copied to the copy code afterward (online change)
	name : WSTRING;
	parent : TOF_Testing.ITestElement;
	scenario : DELAYED_TIMER_TEST_SCENARIO;
END_VAR
_Scenario := scenario;
_Timeout := T#10S;
FB_init := TRUE;
END_METHOD

(*!
<summary>Starts the positive interval directly or by restarting an already active long timer.</summary>
*)
METHOD PROTECTED BeforeTest
IF _Scenario = DELAYED_TIMER_TEST_SCENARIO.AFTER_ACTIVE_RESTART THEN
	_Timer.Interval := _ActiveInterval;

	IF NOT _Timer.Start() THEN
		RecordFailure(message := "The long timer must start before positive restart");
		RETURN;
	END_IF

	_StartedAt := Tc2_System.F_GetTaskTime();
	Assert.ThatBool(
		actual := _Timer.SetIntervalAndRestart(interval := _PositiveInterval),
		message := "The active timer must restart with a positive preset"
	).IsTrue();
ELSE
	_Timer.Interval := _PositiveInterval;
	_StartedAt := Tc2_System.F_GetTaskTime();
	Assert.ThatBool(actual := _Timer.Start(), message := "The prepared positive timer must accept Start").IsTrue();
END_IF
END_METHOD

(*!
<summary>Waits without evaluating TON, then observes completion or requested cancellation.</summary>
*)
METHOD PROTECTED ExecuteTest : TOF_Testing.TEST_CYCLE_RESULT
VAR
	currentTaskTime : ULINT;
	elapsedTicks : ULINT;
END_VAR
ExecuteTest := TOF_Testing.TEST_CYCLE_RESULT.DONE;
currentTaskTime := Tc2_System.F_GetTaskTime();

IF currentTaskTime < _StartedAt THEN
	RecordFailure(message := "Independent task time moved backwards");
	RETURN;
END_IF

elapsedTicks := currentTaskTime - _StartedAt;
Assert.ThatBool(
	actual := _Timer.State.Running,
	message := "The timer must remain running until its first Execute"
).IsTrue();
Assert.ThatBool(
	actual := _Timer.Elapsed,
	message := "Skipping Execute must preserve the unelapsed observation"
).IsFalse();
Assert.ThatBool(
	actual := _Timer.ElapsedTime = TOF_Core.Times.MIN_VALUE,
	message := "Getter reads must leave elapsed time at zero before the first Execute"
).IsTrue();

IF elapsedTicks < TO_ULINT(_PositiveInterval) * _TaskTimeTicksPerMillisecond + _TimingToleranceTicks THEN
	ExecuteTest := TOF_Testing.TEST_CYCLE_RESULT.BUSY;
	RETURN;
END_IF

IF Outcome = TOF_Testing.TEST_OUTCOME.FAILED THEN
	RETURN;
END_IF

IF _Scenario = DELAYED_TIMER_TEST_SCENARIO.CANCEL_BEFORE_EXECUTE THEN
	IF NOT _Timer.Cancel() THEN
		RecordFailure(message := "Cancel must take precedence over unobserved expiry");
		RETURN;
	END_IF

	_Timer.Execute();
	Assert.ThatBool(
		actual := _Timer.State.Stopped,
		message := "Cancellation must finish on the first Execute"
	).IsTrue();
	Assert.ThatBool(
		actual := _Timer.FinalStopReason.ExternalCancel,
		message := "Unobserved expiry must not replace cancellation"
	).IsTrue();
	Assert.ThatBool(
		actual := _Timer.Triggered,
		message := "Cancelled unobserved expiry must not trigger"
	).IsFalse();
	Assert.ThatBool(
		actual := _Timer.Elapsed,
		message := "Stopping must leave the unobserved TON expiry unevaluated"
	).IsFalse();
	Assert.ThatBool(
		actual := _Timer.ElapsedTime = TOF_Core.Times.MIN_VALUE,
		message := "Unobserved cancellation must preserve zero elapsed time"
	).IsTrue();

	RETURN;
END_IF

_Timer.Execute();
Assert.ThatBool(
	actual := _Timer.Triggered,
	message := "The first delayed Execute must observe expiry anchored at Start"
).IsTrue();
Assert.ThatBool(actual := _Timer.Elapsed, message := "Delayed completion must expose TON.Q").IsTrue();
Assert.ThatBool(actual := _Timer.State.Stopped, message := "Delayed completion must be immediate").IsTrue();
Assert.ThatBool(
	actual := _Timer.FinalStopReason.WorkDone,
	message := "Delayed completion must remain successful"
).IsTrue();
Assert.ThatBool(
	actual := _Timer.ElapsedTime = _PositiveInterval,
	message := "Completed elapsed time must reach the positive preset"
).IsTrue();

IF Outcome = TOF_Testing.TEST_OUTCOME.FAILED THEN
	RETURN;
END_IF

IF NOT _Timer.SetIntervalAndRestart(interval := _PositiveInterval) THEN
	RecordFailure(message := "A completed positive timer must accept positive restart");
	RETURN;
END_IF

Assert.ThatBool(
	actual := _Timer.State.Running,
	message := "Positive restart must start a new run immediately"
).IsTrue();
Assert.ThatBool(actual := _Timer.Elapsed, message := "Positive restart must clear the prior Q").IsFalse();
Assert.ThatBool(
	actual := _Timer.Triggered,
	message := "Positive restart must clear the prior completion pulse"
).IsFalse();
Assert.ThatBool(
	actual := _Timer.Cancel(),
	message := "The active replacement run must accept cancellation"
).IsTrue();
_Timer.Execute();
Assert.ThatBool(
	actual := _Timer.State.Stopped AND_THEN _Timer.FinalStopReason.ExternalCancel,
	message := "The replacement run must finish cancellation"
).IsTrue();
END_METHOD

(*!
<summary>Returns the owned timer to READY before reporting the result.</summary>
<description>
Cooperatively cancels active work and clears any retained TON observations through Reset.
</description>
*)
METHOD PROTECTED AfterTest
Assert.ThatBool(
	actual := PrepareTimerTestForReuse(timer := _Timer),
	message := "The timer must return to READY after cleanup"
).IsTrue();
END_METHOD

//! <summary>Borrows the concrete class name. Callers must not modify it.</summary>
{attribute 'monitoring' := 'call'}
PROPERTY ClassName : REFERENCE TO STRING
GET
ClassName REF= _ClassName;
END_GET
END_PROPERTY

//! <summary>Borrows the compiler-initialized namespace. Callers must not modify it.</summary>
{attribute 'monitoring' := 'call'}
PROPERTY NamespaceName : REFERENCE TO STRING
GET
NamespaceName REF= CurrentNamespace.Name;
END_GET
END_PROPERTY

//! <summary>Reports the concrete instance size in bytes.</summary>
{attribute 'monitoring' := 'call'}
PROPERTY SelfSize : ULINT
GET
SelfSize := XSIZEOF(THIS^);
END_GET
END_PROPERTY

END_FUNCTION_BLOCK

// ---- Tests/Tasks/Stopping/TaskStoppingTestGroup.TcPOU
(*
SPDX-FileCopyrightText: © 2026 Oleksandr Tiutyk <trofimich@gmail.com>
SPDX-License-Identifier: MIT
License: https://opensource.org/license/mit
*)

(*!
<summary>Groups the cooperative stopping, failure and task naming tests.</summary>
<description>
Owns independent fixtures and the fixed child array. Use from one PLC task and keep the group at a stable address.
</description>
*)

{attribute 'no_assign'}
{attribute 'no_explicit_call' := 'do not call this function block directly'}
FUNCTION_BLOCK TaskStoppingTestGroup EXTENDS TOF_Testing.TestGroup<17>
VAR_STAT
	{attribute 'hide'}
	_ClassName : STRING := __POUNAME();
END_VAR
VAR
	_NameBeforeStartAndAfterReset : TaskStoppingNameTest(
		name := "NameBeforeStartAndAfterReset",
		parent := THIS^
	);
	_SuccessWaitsForCleanup : TaskStoppingScenarioTest(
		name := "SuccessWaitsForCleanup",
		parent := THIS^,
		scenario := TASK_STOPPING_TEST_SCENARIO.WORK_DONE
	);
	_ErrorWaitsForCleanup : TaskStoppingScenarioTest(
		name := "ErrorWaitsForCleanup",
		parent := THIS^,
		scenario := TASK_STOPPING_TEST_SCENARIO.WORK_ERROR
	);
	_AbortWaitsForCleanup : TaskStoppingScenarioTest(
		name := "AbortWaitsForCleanup",
		parent := THIS^,
		scenario := TASK_STOPPING_TEST_SCENARIO.WORK_ABORT
	);
	_ExceptionWaitsForCleanup : TaskStoppingScenarioTest(
		name := "ExceptionWaitsForCleanup",
		parent := THIS^,
		scenario := TASK_STOPPING_TEST_SCENARIO.WORK_EXCEPTION
	);
	_FormattingFailureWaitsForCleanup : TaskStoppingScenarioTest(
		name := "FormattingFailureWaitsForCleanup",
		parent := THIS^,
		scenario := TASK_STOPPING_TEST_SCENARIO.WORK_FORMATTER_EXCEPTION
	);
	_StoppingExceptionResumes : TaskStoppingScenarioTest(
		name := "StoppingExceptionResumes",
		parent := THIS^,
		scenario := TASK_STOPPING_TEST_SCENARIO.FIRST_STOPPING_EXCEPTION
	);
	_RepeatedStoppingExceptions : TaskStoppingScenarioTest(
		name := "RepeatedStoppingExceptions",
		parent := THIS^,
		scenario := TASK_STOPPING_TEST_SCENARIO.REPEATED_STOPPING_EXCEPTIONS
	);
	_EmptyExceptionMessageUsesFallback : TaskStoppingScenarioTest(
		name := "EmptyExceptionMessageUsesFallback",
		parent := THIS^,
		scenario := TASK_STOPPING_TEST_SCENARIO.EMPTY_WORK_EXCEPTION_MESSAGE
	);
	_CancelDuringAcquire : TaskStoppingScenarioTest(
		name := "CancelDuringAcquire",
		parent := THIS^,
		scenario := TASK_STOPPING_TEST_SCENARIO.CANCEL_DURING_ACQUIRE
	);
	_CancelBeforeAcquire : TaskStoppingScenarioTest(
		name := "CancelBeforeAcquire",
		parent := THIS^,
		scenario := TASK_STOPPING_TEST_SCENARIO.CANCEL_BEFORE_ACQUIRE
	);
	_AcquireFailureWithResource : TaskStoppingScenarioTest(
		name := "AcquireFailureWithResource",
		parent := THIS^,
		scenario := TASK_STOPPING_TEST_SCENARIO.ACQUIRE_EXCEPTION_AFTER_OWNERSHIP
	);
	_AcquireFailureWithoutResource : TaskStoppingScenarioTest(
		name := "AcquireFailureWithoutResource",
		parent := THIS^,
		scenario := TASK_STOPPING_TEST_SCENARIO.ACQUIRE_EXCEPTION_BEFORE_OWNERSHIP
	);
	_ReleaseFailurePreservesOriginal : TaskStoppingScenarioTest(
		name := "ReleaseFailurePreservesOriginal",
		parent := THIS^,
		scenario := TASK_STOPPING_TEST_SCENARIO.RELEASE_EXCEPTION
	);
	_ResetFromAfterStop : TaskStoppingScenarioTest(
		name := "ResetFromAfterStop",
		parent := THIS^,
		scenario := TASK_STOPPING_TEST_SCENARIO.RESET_IN_NOTIFICATION
	);
	_ResetFormattingFailure : TaskStoppingScenarioTest(
		name := "ResetFormattingFailure",
		parent := THIS^,
		scenario := TASK_STOPPING_TEST_SCENARIO.RESET_FORMATTER_EXCEPTION
	);
	_StartFormattingFailure : TaskStoppingScenarioTest(
		name := "StartFormattingFailure",
		parent := THIS^,
		scenario := TASK_STOPPING_TEST_SCENARIO.START_FORMATTER_EXCEPTION
	);

	_Children : ARRAY [0.._ChildCount - 1] OF TOF_Testing.ITestElement :=
	[
		_NameBeforeStartAndAfterReset,
		_SuccessWaitsForCleanup,
		_ErrorWaitsForCleanup,
		_AbortWaitsForCleanup,
		_ExceptionWaitsForCleanup,
		_FormattingFailureWaitsForCleanup,
		_StoppingExceptionResumes,
		_RepeatedStoppingExceptions,
		_EmptyExceptionMessageUsesFallback,
		_CancelDuringAcquire,
		_CancelBeforeAcquire,
		_AcquireFailureWithResource,
		_AcquireFailureWithoutResource,
		_ReleaseFailurePreservesOriginal,
		_ResetFromAfterStop,
		_ResetFormattingFailure,
		_StartFormattingFailure
	];
END_VAR

//! <summary>Borrows the fixed child array. Callers must not modify it.</summary>
{attribute 'monitoring' := 'call'}
PROPERTY Children : REFERENCE TO ARRAY [0.._ChildCount - 1] OF TOF_Testing.ITestElement
GET
Children REF= _Children;
END_GET
END_PROPERTY

//! <summary>Borrows the concrete class name. Callers must not modify it.</summary>
{attribute 'monitoring' := 'call'}
PROPERTY ClassName : REFERENCE TO STRING
GET
ClassName REF= _ClassName;
END_GET
END_PROPERTY

//! <summary>Borrows the compiler-initialized namespace name. Callers must not modify it.</summary>
{attribute 'monitoring' := 'call'}
PROPERTY NamespaceName : REFERENCE TO STRING
GET
NamespaceName REF= CurrentNamespace.Name;
END_GET
END_PROPERTY

//! <summary>Reports the concrete instance size in bytes.</summary>
{attribute 'monitoring' := 'call'}
PROPERTY SelfSize : ULINT
GET
SelfSize := XSIZEOF(THIS^);
END_GET
END_PROPERTY

END_FUNCTION_BLOCK

// ---- Tests/Tasks/Stopping/TaskStoppingNameTest.TcPOU
(*
SPDX-FileCopyrightText: © 2026 Oleksandr Tiutyk <trofimich@gmail.com>
SPDX-License-Identifier: MIT
License: https://opensource.org/license/mit
*)

(*!
<summary>Checks default and explicit names through the task lifecycle.</summary>
<description>
Drives a probe without external resources. The instance retains borrowed name storage across Execute and Reset.
</description>
*)

{attribute 'no_assign'}
{attribute 'no_explicit_call' := 'do not call this function block directly'}
FUNCTION_BLOCK TaskStoppingNameTest EXTENDS TOF_Testing.MultiCycleTest
VAR_STAT
	{attribute 'hide'}
	_ClassName : STRING := __POUNAME();
END_VAR
VAR
	_Task : TaskStoppingProbe(name := "");
	_NamedTask : TaskStoppingProbe(name := "Named stopping probe");
	_InitialName : WSTRING;
	_BorrowedName : REFERENCE TO WSTRING;
END_VAR

(*!
<summary>Reads and retains the default name before starting resource-free work.</summary>
*)
METHOD PROTECTED BeforeTest
_BorrowedName REF= _Task.Name;

IF NOT __ISVALIDREF(_BorrowedName) THEN
	RecordFailure(message := "Default name must be available before Start");
	RETURN;
END_IF

_InitialName := _BorrowedName;
Assert.ThatWideString(
	actual := Tc2_Standard.WLEFT(STR := _InitialName, SIZE := Tc2_Standard.WLEN(STR := "TaskStoppingProbe")),
	message := "Default name must include the initialized concrete class"
).ToBe(expected := "TaskStoppingProbe");
Assert.ThatWideString(
	actual := _NamedTask.Name,
	message := "Explicit name must survive construction"
).ToBe(expected := "Named stopping probe");
Assert.ThatWideString(
	actual := _Task.Name,
	message := "Repeated reads must preserve the name"
).ToBe(expected := _InitialName);
Assert.ThatBool(actual := _Task.State.Ready, message := "Reading Name must not start the task").IsTrue();

IF Outcome = TOF_Testing.TEST_OUTCOME.FAILED THEN
	RETURN;
END_IF

Assert.ThatBool(actual := _Task.Start(), message := "Prepared probe must accept Start").IsTrue();
END_METHOD

(*!
<summary>Checks the same name during execution and the borrowed address after Reset.</summary>
*)
METHOD PROTECTED ExecuteTest : TOF_Testing.TEST_CYCLE_RESULT
VAR
	nameAfterReset : REFERENCE TO WSTRING;
END_VAR
_Task.Execute();
Assert.ThatWideString(
	actual := _Task.Name,
	message := "Lifecycle progress must preserve the name"
).ToBe(expected := _InitialName);

IF NOT _Task.State.Stopped THEN
	ExecuteTest := TOF_Testing.TEST_CYCLE_RESULT.BUSY;
	RETURN;
END_IF

ExecuteTest := TOF_Testing.TEST_CYCLE_RESULT.DONE;

IF NOT _Task.Reset() THEN
	RecordFailure(message := "Completed probe must accept Reset");
	RETURN;
END_IF

nameAfterReset REF= _Task.Name;

IF NOT __ISVALIDREF(nameAfterReset) OR_ELSE NOT __ISVALIDREF(_BorrowedName) THEN
	RecordFailure(message := "Both name references must remain valid after Reset");
	RETURN;
END_IF

Assert.ThatBool(
	actual := ADR(nameAfterReset) = ADR(_BorrowedName),
	message := "Reset must preserve the address of borrowed name storage"
).IsTrue();
Assert.ThatWideString(
	actual := nameAfterReset,
	message := "Reset must preserve the name text"
).ToBe(expected := _InitialName);
END_METHOD

(*!
<summary>Clears the borrowed name and completes up to two remaining resource-free stopping steps.</summary>
*)
METHOD PROTECTED AfterTest
_BorrowedName REF= 0;

IF _Task.State.Running THEN
	IF NOT _Task.OriginalStopReason.ExternalCancel THEN
		_Task.Cancel();
	END_IF

	// The probe has two synthetic cleanup steps and no bound resource.
	_Task.Execute();

	IF _Task.State.Running THEN
		_Task.Execute();
	END_IF
END_IF

IF _Task.State.Stopped THEN
	Assert.ThatBool(actual := _Task.Reset(), message := "The name probe must accept cleanup Reset").IsTrue();
END_IF

Assert.ThatBool(actual := _Task.State.Ready, message := "The name probe must be READY after cleanup").IsTrue();
END_METHOD

//! <summary>Borrows the concrete class name. Callers must not modify it.</summary>
{attribute 'monitoring' := 'call'}
PROPERTY ClassName : REFERENCE TO STRING
GET
ClassName REF= _ClassName;
END_GET
END_PROPERTY

//! <summary>Borrows the compiler-initialized namespace name. Callers must not modify it.</summary>
{attribute 'monitoring' := 'call'}
PROPERTY NamespaceName : REFERENCE TO STRING
GET
NamespaceName REF= CurrentNamespace.Name;
END_GET
END_PROPERTY

//! <summary>Reports the concrete instance size in bytes.</summary>
{attribute 'monitoring' := 'call'}
PROPERTY SelfSize : ULINT
GET
SelfSize := XSIZEOF(THIS^);
END_GET
END_PROPERTY

END_FUNCTION_BLOCK

// ---- Tests/Tasks/Stopping/TaskStoppingProbe.TcPOU
(*
SPDX-FileCopyrightText: © 2026 Oleksandr Tiutyk <trofimich@gmail.com>
SPDX-License-Identifier: MIT
License: https://opensource.org/license/mit
*)

(*!
<summary>Exercises the production Task lifecycle with delayed, interruptible stopping.</summary>
<description>
The scenario owns and injects a TaskStoppingResource through SetResource before Start. The binding is borrowed
and stable across runs. Inputs configure faults; ThrowOnEveryStopping may be cleared while RUNNING to resume
cleanup. Observations are cumulative until ClearObservations, except cleanup progress, which OnReset clears.
No physical I/O is performed.
</description>
*)

